    |   movel([0.069164, -1.303567, -2.624691, -0.784131, 1.570796, 1.639960],accel_mss,speed_ms,0,blend_radius_m)
    |   movel([0.068809, -1.303606, -2.624668, -0.784115, 1.570796, 1.639606],accel_mss,speed_ms,0,blend_radius_m)
    |   movel([0.068472, -1.303670, -2.624630, -0.784090, 1.570796, 1.639268],accel_mss,speed_ms,0,blend_radius_m)
    |   movel([0.068228, -1.303624, -2.624657, -0.784108, 1.570796, 1.639025],accel_mss,speed_ms,0,blend_radius_m)
    |   movel([0.068160, -1.303397, -2.624793, -0.784199, 1.570796, 1.638957],accel_mss,speed_ms,0,blend_radius_m)
    |   movel([0.067957, -1.303250, -2.624881, -0.784258, 1.570796, 1.638753],accel_mss,speed_ms,0,blend_radius_m)
    |   movel([0.067920, -1.302997, -2.625033, -0.784360, 1.570796, 1.638717],accel_mss,speed_ms,0,blend_radius_m)
    |   movel([0.068076, -1.302591, -2.625275, -0.784523, 1.570796, 1.638872],accel_mss,speed_ms,0,blend_radius_m)
    |   movel([0.068245, -1.302321, -2.625436, -0.784631, 1.570796, 1.639041],accel_mss,speed_ms,0,blend_radius_m)
    |   movel([0.068538, -1.301870, -2.625706, -0.784813, 1.570796, 1.639334],accel_mss,speed_ms,0,blend_radius_m)
    |   movel([0.068564, -1.301570, -2.625885, -0.784934, 1.570796, 1.639361],accel_mss,speed_ms,0,blend_radius_m)
    |   movel([0.068351, -1.301410, -2.625980, -0.784999, 1.570796, 1.639147],accel_mss,speed_ms,0,blend_radius_m)
    |   movel([0.068159, -1.301249, -2.626076, -0.785063, 1.570796, 1.638955],accel_mss,speed_ms,0,blend_radius_m)
    |   movel([0.068070, -1.301051, -2.626194, -0.785144, 1.570796, 1.638866],accel_mss,speed_ms,0,blend_radius_m)
    |   movel([0.067838, -1.300944, -2.626258, -0.785187, 1.570796, 1.638635],accel_mss,speed_ms,0,blend_radius_m)
    |   movel([0.067733, -1.300746, -2.626376, -0.785267, 1.570796, 1.638529],accel_mss,speed_ms,0,blend_radius_m)
    |   movel([0.067965, -1.300491, -2.626528, -0.785370, 1.570796, 1.638762],accel_mss,speed_ms,0,blend_radius_m)
    |   movel([0.068177, -1.300786, -2.626352, -0.785251, 1.570796, 1.638973],accel_mss,speed_ms,0,blend_radius_m)
    |   movel([0.068448, -1.300963, -2.626247, -0.785179, 1.570796, 1.639244],accel_mss,speed_ms,0,blend_radius_m)
    |   movel([0.068582, -1.300695, -2.626406, -0.785288, 1.570796, 1.639379],accel_mss,speed_ms,0,blend_radius_m)
    |   movel([0.068570, -1.300446, -2.626554, -0.785388, 1.570796, 1.639366],accel_mss,speed_ms,0,blend_radius_m)
    |   movel([0.068283, -1.300598, -2.626464, -0.785327, 1.570796, 1.639079],accel_mss,speed_ms,0,blend_radius_m)
    |   movel([0.068322, -1.300335, -2.626620, -0.785433, 1.570796, 1.639119],accel_mss,speed_ms,0,blend_radius_m)
    |   movel([0.068410, -1.300077, -2.626774, -0.785538, 1.570796, 1.639206],accel_mss,speed_ms,0,blend_radius_m)
    |   movel([0.068413, -1.299834, -2.626919, -0.785637, 1.570796, 1.639209],accel_mss,speed_ms,0,blend_radius_m)
    |   movel([0.068610, -1.299527, -2.627101, -0.785761, 1.570796, 1.639406],accel_mss,speed_ms,0,blend_radius_m)
    |   movel([0.068344, -1.299545, -2.627090, -0.785754, 1.570796, 1.639140],accel_mss,speed_ms,0,blend_radius_m)
    |   movel([0.068247, -1.299852, -2.626908, -0.785629, 1.570796, 1.639043],accel_mss,speed_ms,0,blend_radius_m)
    |   movel([0.068015, -1.299788, -2.626946, -0.785655, 1.570796, 1.638811],accel_mss,speed_ms,0,blend_radius_m)
    |   movel([0.068098, -1.299347, -2.627208, -0.785834, 1.570796, 1.638894],accel_mss,speed_ms,0,blend_radius_m)
    |   movel([0.068346, -1.299039, -2.627391, -0.785960, 1.570796, 1.639142],accel_mss,speed_ms,0,blend_radius_m)
    |   movel([0.068703, -1.298720, -2.627579, -0.786089, 1.570796, 1.639499],accel_mss,speed_ms,0,blend_radius_m)
    |   movel([0.069005, -1.298409, -2.627764, -0.786216, 1.570796, 1.639802],accel_mss,speed_ms,0,blend_radius_m)
    |   movel([0.068736, -1.297952, -2.628034, -0.786402, 1.570796, 1.639533],accel_mss,speed_ms,0,blend_radius_m)
    |   movel([0.068447, -1.297686, -2.628192, -0.786511, 1.570796, 1.639243],accel_mss,speed_ms,0,blend_radius_m)
    |   movel([0.068186, -1.297495, -2.628305, -0.786589, 1.570796, 1.638982],accel_mss,speed_ms,0,blend_radius_m)
    |   movel([0.068055, -1.297206, -2.628475, -0.786707, 1.570796, 1.638851],accel_mss,speed_ms,0,blend_radius_m)
    |   movel([0.068400, -1.296905, -2.628653, -0.786831, 1.570796, 1.639196],accel_mss,speed_ms,0,blend_radius_m)
    |   movel([0.068673, -1.296731, -2.628756, -0.786902, 1.570796, 1.639470],accel_mss,speed_ms,0,blend_radius_m)
    |   movel([0.068591, -1.296502, -2.628891, -0.786996, 1.570796, 1.639387],accel_mss,speed_ms,0,blend_radius_m)
    |   movel([0.068494, -1.296286, -2.629019, -0.787084, 1.570796, 1.639291],accel_mss,speed_ms,0,blend_radius_m)
    |   movel([0.068508, -1.296042, -2.629162, -0.787184, 1.570796, 1.639305],accel_mss,speed_ms,0,blend_radius_m)
    |   movel([0.068313, -1.295946, -2.629219, -0.787224, 1.570796, 1.639109],accel_mss,speed_ms,0,blend_radius_m)
    |   movel([0.068432, -1.295566, -2.629443, -0.787380, 1.570796, 1.639228],accel_mss,speed_ms,0,blend_radius_m)
    |   movel([0.068734, -1.295104, -2.629715, -0.787570, 1.570796, 1.639530],accel_mss,speed_ms,0,blend_radius_m)
    |   movel([0.069080, -1.294873, -2.629850, -0.787665, 1.570796, 1.639876],accel_mss,speed_ms,0,blend_radius_m)
    |   movel([0.069351, -1.294697, -2.629954, -0.787738, 1.570796, 1.640148],accel_mss,speed_ms,0,blend_radius_m)
    |   movel([0.069675, -1.294448, -2.630100, -0.787841, 1.570796, 1.640471],accel_mss,speed_ms,0,blend_radius_m)
    |   movel([0.069973, -1.294347, -2.630159, -0.787882, 1.570796, 1.640769],accel_mss,speed_ms,0,blend_radius_m)
    |   movel([0.070329, -1.294063, -2.630326, -0.788000, 1.570796, 1.641125],accel_mss,speed_ms,0,blend_radius_m)
    |   movel([0.070734, -1.293918, -2.630411, -0.788060, 1.570796, 1.641530],accel_mss,speed_ms,0,blend_radius_m)
    |   movel([0.070848, -1.294112, -2.630297, -0.787979, 1.570796, 1.641644],accel_mss,speed_ms,0,blend_radius_m)
    |   movel([0.070586, -1.294072, -2.630321, -0.787996, 1.570796, 1.641382],accel_mss,speed_ms,0,blend_radius_m)
    |   movel([0.070545, -1.294342, -2.630162, -0.787884, 1.570796, 1.641341],accel_mss,speed_ms,0,blend_radius_m)
    |   movel([0.070287, -1.294320, -2.630176, -0.787894, 1.570796, 1.641083],accel_mss,speed_ms,0,blend_radius_m)
    |   movel([0.070092, -1.294585, -2.630020, -0.787784, 1.570796, 1.640888],accel_mss,speed_ms,0,blend_radius_m)
    |   movel([0.069788, -1.294730, -2.629935, -0.787724, 1.570796, 1.640584],accel_mss,speed_ms,0,blend_radius_m)
    |   movel([0.070023, -1.294763, -2.629915, -0.787711, 1.570796, 1.640820],accel_mss,speed_ms,0,blend_radius_m)
    |   movel([0.070448, -1.294538, -2.630047, -0.787804, 1.570796, 1.641244],accel_mss,speed_ms,0,blend_radius_m)
    |   movel([0.070733, -1.294397, -2.630130, -0.787862, 1.570796, 1.641529],accel_mss,speed_ms,0,blend_radius_m)
    |   movel([0.071014, -1.294267, -2.630206, -0.787915, 1.570796, 1.641811],accel_mss,speed_ms,0,blend_radius_m)
    |   movel([0.071419, -1.294059, -2.630329, -0.788002, 1.570796, 1.642215],accel_mss,speed_ms,0,blend_radius_m)
    |   movel([0.071699, -1.293711, -2.630533, -0.788145, 1.570796, 1.642496],accel_mss,speed_ms,0,blend_radius_m)
    |   movel([0.071397, -1.293860, -2.630445, -0.788084, 1.570796, 1.642193],accel_mss,speed_ms,0,blend_radius_m)
    |   movel([0.071394, -1.293531, -2.630638, -0.788220, 1.570796, 1.642190],accel_mss,speed_ms,0,blend_radius_m)
    |   movel([0.071674, -1.293324, -2.630760, -0.788306, 1.570796, 1.642471],accel_mss,speed_ms,0,blend_radius_m)
    |   movel([0.072099, -1.293139, -2.630868, -0.788382, 1.570796, 1.642895],accel_mss,speed_ms,0,blend_radius_m)
    |   movel([0.072618, -1.292956, -2.630975, -0.788458, 1.570796, 1.643415],accel_mss,speed_ms,0,blend_radius_m)
    |   movel([0.072298, -1.293292, -2.630778, -0.788319, 1.570796, 1.643094],accel_mss,speed_ms,0,blend_radius_m)
    |   movel([0.072072, -1.293569, -2.630616, -0.788204, 1.570796, 1.642868],accel_mss,speed_ms,0,blend_radius_m)
    |   movel([0.072318, -1.293598, -2.630599, -0.788192, 1.570796, 1.643115],accel_mss,speed_ms,0,blend_radius_m)
    |   movel([0.072810, -1.293423, -2.630701, -0.788264, 1.570796, 1.643606],accel_mss,speed_ms,0,blend_radius_m)
    |   movel([0.073098, -1.293441, -2.630691, -0.788257, 1.570796, 1.643895],accel_mss,speed_ms,0,blend_radius_m)
    |   movel([0.073371, -1.293396, -2.630718, -0.788276, 1.570796, 1.644167],accel_mss,speed_ms,0,blend_radius_m)
    |   movel([0.073643, -1.293184, -2.630842, -0.788364, 1.570796, 1.644439],accel_mss,speed_ms,0,blend_radius_m)
    |   movel([0.073422, -1.293074, -2.630906, -0.788409, 1.570796, 1.644218],accel_mss,speed_ms,0,blend_radius_m)
    |   movel([0.073605, -1.292634, -2.631163, -0.788592, 1.570796, 1.644402],accel_mss,speed_ms,0,blend_radius_m)
    |   movel([0.074088, -1.292377, -2.631314, -0.788698, 1.570796, 1.644884],accel_mss,speed_ms,0,blend_radius_m)
    |   movel([0.074586, -1.292293, -2.631363, -0.788733, 1.570796, 1.645382],accel_mss,speed_ms,0,blend_radius_m)
    |   movel([0.075419, -1.292221, -2.631405, -0.788763, 1.570796, 1.646216],accel_mss,speed_ms,0,blend_radius_m)
    |   movel([0.075774, -1.292192, -2.631422, -0.788775, 1.570796, 1.646570],accel_mss,speed_ms,0,blend_radius_m)
    |   movel([0.076162, -1.292154, -2.631444, -0.788791, 1.570796, 1.646959],accel_mss,speed_ms,0,blend_radius_m)
    |   movel([0.076529, -1.292117, -2.631466, -0.788806, 1.570796, 1.647325],accel_mss,speed_ms,0,blend_radius_m)
    |   movel([0.076800, -1.292084, -2.631485, -0.788820, 1.570796, 1.647596],accel_mss,speed_ms,0,blend_radius_m)
    |   movel([0.077294, -1.292079, -2.631488, -0.788822, 1.570796, 1.648090],accel_mss,speed_ms,0,blend_radius_m)
    |   movel([0.077690, -1.292165, -2.631437, -0.788786, 1.570796, 1.648486],accel_mss,speed_ms,0,blend_radius_m)
    |   movel([0.078122, -1.292360, -2.631324, -0.788705, 1.570796, 1.648918],accel_mss,speed_ms,0,blend_radius_m)
    |   movel([0.078432, -1.292469, -2.631260, -0.788660, 1.570796, 1.649228],accel_mss,speed_ms,0,blend_radius_m)
    |   movel([0.078708, -1.292526, -2.631227, -0.788636, 1.570796, 1.649504],accel_mss,speed_ms,0,blend_radius_m)
    |   movel([0.079022, -1.292550, -2.631212, -0.788626, 1.570796, 1.649819],accel_mss,speed_ms,0,blend_radius_m)
    |   movel([0.079477, -1.292643, -2.631158, -0.788588, 1.570796, 1.650273],accel_mss,speed_ms,0,blend_radius_m)
    |   movel([0.080017, -1.292922, -2.630995, -0.788472, 1.570796, 1.650813],accel_mss,speed_ms,0,blend_radius_m)
    |   movel([0.080490, -1.293278, -2.630787, -0.788325, 1.570796, 1.651286],accel_mss,speed_ms,0,blend_radius_m)
    |   movel([0.080723, -1.293620, -2.630586, -0.788183, 1.570796, 1.651519],accel_mss,speed_ms,0,blend_radius_m)
    |   movel([0.080790, -1.293977, -2.630377, -0.788035, 1.570796, 1.651586],accel_mss,speed_ms,0,blend_radius_m)
    |   movel([0.080755, -1.294421, -2.630116, -0.787852, 1.570796, 1.651551],accel_mss,speed_ms,0,blend_radius_m)
    |   movel([0.080623, -1.294881, -2.629846, -0.787662, 1.570796, 1.651420],accel_mss,speed_ms,0,blend_radius_m)
    |   movel([0.080414, -1.295282, -2.629610, -0.787497, 1.570796, 1.651210],accel_mss,speed_ms,0,blend_radius_m)
    |   movel([0.080193, -1.295571, -2.629440, -0.787378, 1.570796, 1.650990],accel_mss,speed_ms,0,blend_radius_m)
    |   movel([0.079916, -1.295860, -2.629270, -0.787259, 1.570796, 1.650712],accel_mss,speed_ms,0,blend_radius_m)
    |   movel([0.079600, -1.296134, -2.629108, -0.787147, 1.570796, 1.650396],accel_mss,speed_ms,0,blend_radius_m)
    |   movel([0.079260, -1.296379, -2.628964, -0.787046, 1.570796, 1.650056],accel_mss,speed_ms,0,blend_radius_m)
    |   movel([0.079132, -1.296209, -2.629064, -0.787116, 1.570796, 1.649929],accel_mss,speed_ms,0,blend_radius_m)
    |   movel([0.078790, -1.296573, -2.628849, -0.786967, 1.570796, 1.649586],accel_mss,speed_ms,0,blend_radius_m)
    |   movel([0.078548, -1.296803, -2.628714, -0.786872, 1.570796, 1.649345],accel_mss,speed_ms,0,blend_radius_m)
    |   movel([0.078210, -1.297243, -2.628454, -0.786692, 1.570796, 1.649006],accel_mss,speed_ms,0,blend_radius_m)
    |   movel([0.078166, -1.297522, -2.628289, -0.786578, 1.570796, 1.648962],accel_mss,speed_ms,0,blend_radius_m)
    |   movel([0.078357, -1.297855, -2.628092, -0.786442, 1.570796, 1.649153],accel_mss,speed_ms,0,blend_radius_m)
    |   movel([0.078391, -1.298108, -2.627942, -0.786339, 1.570796, 1.649187],accel_mss,speed_ms,0,blend_radius_m)
    |   movel([0.078328, -1.298389, -2.627776, -0.786224, 1.570796, 1.649124],accel_mss,speed_ms,0,blend_radius_m)
    |   movel([0.078048, -1.298815, -2.627523, -0.786051, 1.570796, 1.648844],accel_mss,speed_ms,0,blend_radius_m)
    |   movel([0.078070, -1.299052, -2.627382, -0.785954, 1.570796, 1.648866],accel_mss,speed_ms,0,blend_radius_m)
    |   movel([0.077797, -1.299433, -2.627156, -0.785799, 1.570796, 1.648593],accel_mss,speed_ms,0,blend_radius_m)
    |   movel([0.077543, -1.299716, -2.626989, -0.785685, 1.570796, 1.648340],accel_mss,speed_ms,0,blend_radius_m)
    |   movel([0.077141, -1.299955, -2.626847, -0.785588, 1.570796, 1.647937],accel_mss,speed_ms,0,blend_radius_m)
    |   movel([0.076881, -1.300164, -2.626722, -0.785503, 1.570796, 1.647677],accel_mss,speed_ms,0,blend_radius_m)
    |   movel([0.076380, -1.300334, -2.626621, -0.785434, 1.570796, 1.647176],accel_mss,speed_ms,0,blend_radius_m)
    |   movel([0.076038, -1.301452, -2.625956, -0.784982, 1.570796, 1.646834],accel_mss,speed_ms,0,blend_radius_m)
    |   movel([0.075953, -1.301880, -2.625700, -0.784809, 1.570796, 1.646749],accel_mss,speed_ms,0,blend_radius_m)
    |   movel([0.075814, -1.302178, -2.625522, -0.784689, 1.570796, 1.646610],accel_mss,speed_ms,0,blend_radius_m)
    |   movel([0.075570, -1.302494, -2.625333, -0.784562, 1.570796, 1.646366],accel_mss,speed_ms,0,blend_radius_m)
    |   movel([0.075189, -1.302835, -2.625129, -0.784425, 1.570796, 1.645986],accel_mss,speed_ms,0,blend_radius_m)
    |   movel([0.074854, -1.302969, -2.625049, -0.784371, 1.570796, 1.645650],accel_mss,speed_ms,0,blend_radius_m)
    |   movel([0.074612, -1.303200, -2.624911, -0.784278, 1.570796, 1.645408],accel_mss,speed_ms,0,blend_radius_m)
    |   movel([0.074370, -1.303112, -2.624964, -0.784313, 1.570796, 1.645166],accel_mss,speed_ms,0,blend_radius_m)
    |   movel([0.074338, -1.303394, -2.624794, -0.784200, 1.570796, 1.645134],accel_mss,speed_ms,0,blend_radius_m)
    |   movel([0.073982, -1.303545, -2.624704, -0.784140, 1.570796, 1.644779],accel_mss,speed_ms,0,blend_radius_m)
    |   speed_ms = 0.003
    |   movel([0.073982, -1.289735, -2.618173, -0.804481, 1.570796, 1.644779],accel_mss,speed_ms,0,blend_radius_m)
    |   speed_ms = 1.000
    |   movel([0.073982, -1.263429, -2.604724, -0.844235, 1.570796, 1.644779],accel_mss,speed_ms,0,blend_radius_m)
    |   movel([0.076909, -1.251042, -2.611644, -0.849703, 1.570796, 1.647706],accel_mss,speed_ms,0,blend_radius_m)
    |   movel([0.076909, -1.277513, -2.625256, -0.809620, 1.570796, 1.647706],accel_mss,speed_ms,0,blend_radius_m)
    |   speed_ms = 0.003
    |   movel([0.076909, -1.287904, -2.630229, -0.794256, 1.570796, 1.647706],accel_mss,speed_ms,0,blend_radius_m)
    |   speed_ms = 0.007
    |   movel([0.076129, -1.288050, -2.630144, -0.794195, 1.570796, 1.646925],accel_mss,speed_ms,0,blend_radius_m)
    |   movel([0.075299, -1.288083, -2.630125, -0.794181, 1.570796, 1.646095],accel_mss,speed_ms,0,blend_radius_m)
    |   movel([0.074609, -1.288022, -2.630160, -0.794207, 1.570796, 1.645406],accel_mss,speed_ms,0,blend_radius_m)
    |   movel([0.074509, -1.287833, -2.630270, -0.794286, 1.570796, 1.645305],accel_mss,speed_ms,0,blend_radius_m)
    |   movel([0.074808, -1.287539, -2.630440, -0.794409, 1.570796, 1.645604],accel_mss,speed_ms,0,blend_radius_m)
    |   movel([0.075762, -1.287303, -2.630578, -0.794509, 1.570796, 1.646558],accel_mss,speed_ms,0,blend_radius_m)
    |   movel([0.076791, -1.287181, -2.630648, -0.794560, 1.570796, 1.647587],accel_mss,speed_ms,0,blend_radius_m)
    |   movel([0.077546, -1.287262, -2.630601, -0.794526, 1.570796, 1.648343],accel_mss,speed_ms,0,blend_radius_m)
    |   movel([0.077806, -1.287388, -2.630528, -0.794473, 1.570796, 1.648603],accel_mss,speed_ms,0,blend_radius_m)
    |   movel([0.077509, -1.287716, -2.630338, -0.794335, 1.570796, 1.648305],accel_mss,speed_ms,0,blend_radius_m)
    |   movel([0.076909, -1.287904, -2.630229, -0.794256, 1.570796, 1.647706],accel_mss,speed_ms,0,blend_radius_m)
    |   speed_ms = 0.003
    |   movel([0.076909, -1.291425, -2.631870, -0.789094, 1.570796, 1.647706],accel_mss,speed_ms,0,blend_radius_m)
    |   speed_ms = 0.007
    |   movel([0.076129, -1.291571, -2.631785, -0.789034, 1.570796, 1.646925],accel_mss,speed_ms,0,blend_radius_m)
    |   movel([0.075299, -1.291604, -2.631765, -0.789020, 1.570796, 1.646095],accel_mss,speed_ms,0,blend_radius_m)
    |   movel([0.074609, -1.291543, -2.631801, -0.789045, 1.570796, 1.645406],accel_mss,speed_ms,0,blend_radius_m)
    |   movel([0.074509, -1.291354, -2.631911, -0.789124, 1.570796, 1.645305],accel_mss,speed_ms,0,blend_radius_m)
    |   movel([0.074808, -1.291061, -2.632082, -0.789246, 1.570796, 1.645604],accel_mss,speed_ms,0,blend_radius_m)
    |   movel([0.075762, -1.290825, -2.632220, -0.789345, 1.570796, 1.646558],accel_mss,speed_ms,0,blend_radius_m)
    |   movel([0.076791, -1.290704, -2.632290, -0.789395, 1.570796, 1.647587],accel_mss,speed_ms,0,blend_radius_m)
    |   movel([0.077546, -1.290784, -2.632243, -0.789362, 1.570796, 1.648343],accel_mss,speed_ms,0,blend_radius_m)
    |   movel([0.077806, -1.290910, -2.632170, -0.789309, 1.570796, 1.648603],accel_mss,speed_ms,0,blend_radius_m)
    |   movel([0.077509, -1.291238, -2.631979, -0.789172, 1.570796, 1.648305],accel_mss,speed_ms,0,blend_radius_m)
    |   movel([0.076909, -1.291425, -2.631870, -0.789094, 1.570796, 1.647706],accel_mss,speed_ms,0,blend_radius_m)
    |   speed_ms = 0.003
    |   movel([0.076909, -1.277513, -2.625256, -0.809620, 1.570796, 1.647706],accel_mss,speed_ms,0,blend_radius_m)
    |   speed_ms = 1.000
    |   movel([0.076909, -1.251042, -2.611644, -0.849703, 1.570796, 1.647706],accel_mss,speed_ms,0,blend_radius_m)
    |   movel([0.077291, -1.249693, -2.612387, -0.850309, 1.570796, 1.648088],accel_mss,speed_ms,0,blend_radius_m)
    |   movel([0.077291, -1.276182, -2.626016, -0.810191, 1.570796, 1.648088],accel_mss,speed_ms,0,blend_radius_m)
    |   speed_ms = 0.003
    |   movel([0.077291, -1.286581, -2.630996, -0.794812, 1.570796, 1.648088],accel_mss,speed_ms,0,blend_radius_m)
    |   speed_ms = 0.007
    |   movel([0.076492, -1.286619, -2.630974, -0.794796, 1.570796, 1.647288],accel_mss,speed_ms,0,blend_radius_m)
    |   movel([0.075702, -1.286738, -2.630905, -0.794746, 1.570796, 1.646499],accel_mss,speed_ms,0,blend_radius_m)
    |   movel([0.075018, -1.286926, -2.630796, -0.794667, 1.570796, 1.645814],accel_mss,speed_ms,0,blend_radius_m)
    |   movel([0.074481, -1.287038, -2.630731, -0.794620, 1.570796, 1.645277],accel_mss,speed_ms,0,blend_radius_m)
    |   movel([0.074238, -1.286897, -2.630813, -0.794680, 1.570796, 1.645034],accel_mss,speed_ms,0,blend_radius_m)
    |   movel([0.074188, -1.286422, -2.631088, -0.794880, 1.570796, 1.644984],accel_mss,speed_ms,0,blend_radius_m)
    |   movel([0.074355, -1.285032, -2.631890, -0.795466, 1.570796, 1.645151],accel_mss,speed_ms,0,blend_radius_m)
    |   movel([0.074579, -1.283540, -2.632750, -0.796099, 1.570796, 1.645376],accel_mss,speed_ms,0,blend_radius_m)
    |   movel([0.074809, -1.282447, -2.633377, -0.796565, 1.570796, 1.645605],accel_mss,speed_ms,0,blend_radius_m)
    |   movel([0.075052, -1.281644, -2.633838, -0.796908, 1.570796, 1.645848],accel_mss,speed_ms,0,blend_radius_m)
    |   movel([0.075328, -1.281134, -2.634129, -0.797126, 1.570796, 1.646124],accel_mss,speed_ms,0,blend_radius_m)
    |   movel([0.076329, -1.280304, -2.634603, -0.797481, 1.570796, 1.647126],accel_mss,speed_ms,0,blend_radius_m)
    |   movel([0.078074, -1.279627, -2.634990, -0.797772, 1.570796, 1.648871],accel_mss,speed_ms,0,blend_radius_m)
    |   movel([0.079946, -1.279261, -2.635198, -0.797930, 1.570796, 1.650742],accel_mss,speed_ms,0,blend_radius_m)
    |   movel([0.081399, -1.279367, -2.635138, -0.797884, 1.570796, 1.652195],accel_mss,speed_ms,0,blend_radius_m)
    |   movel([0.081937, -1.279667, -2.634967, -0.797755, 1.570796, 1.652733],accel_mss,speed_ms,0,blend_radius_m)
    |   movel([0.082153, -1.280164, -2.634683, -0.797542, 1.570796, 1.652949],accel_mss,speed_ms,0,blend_radius_m)
    |   movel([0.082056, -1.280944, -2.634238, -0.797207, 1.570796, 1.652852],accel_mss,speed_ms,0,blend_radius_m)
    |   movel([0.081621, -1.282158, -2.633543, -0.796688, 1.570796, 1.652417],accel_mss,speed_ms,0,blend_radius_m)
    |   movel([0.081209, -1.283020, -2.633048, -0.796320, 1.570796, 1.652006],accel_mss,speed_ms,0,blend_radius_m)
    |   movel([0.080540, -1.284202, -2.632369, -0.795818, 1.570796, 1.651337],accel_mss,speed_ms,0,blend_radius_m)
    |   movel([0.079825, -1.285365, -2.631699, -0.795326, 1.570796, 1.650622],accel_mss,speed_ms,0,blend_radius_m)
    |   movel([0.079256, -1.286161, -2.631238, -0.794989, 1.570796, 1.650053],accel_mss,speed_ms,0,blend_radius_m)
    |   movel([0.078803, -1.286738, -2.630905, -0.794746, 1.570796, 1.649599],accel_mss,speed_ms,0,blend_radius_m)
    |   movel([0.078012, -1.286628, -2.630968, -0.794793, 1.570796, 1.648808],accel_mss,speed_ms,0,blend_radius_m)
    |   movel([0.077291, -1.286581, -2.630996, -0.794812, 1.570796, 1.648088],accel_mss,speed_ms,0,blend_radius_m)
    |   speed_ms = 0.003
    |   movel([0.077291, -1.290105, -2.632639, -0.789645, 1.570796, 1.648088],accel_mss,speed_ms,0,blend_radius_m)
    |   speed_ms = 0.007
    |   movel([0.076492, -1.290143, -2.632617, -0.789630, 1.570796, 1.647288],accel_mss,speed_ms,0,blend_radius_m)
    |   movel([0.075702, -1.290262, -2.632548, -0.789580, 1.570796, 1.646499],accel_mss,speed_ms,0,blend_radius_m)
    |   movel([0.075018, -1.290449, -2.632439, -0.789502, 1.570796, 1.645814],accel_mss,speed_ms,0,blend_radius_m)
    |   movel([0.074481, -1.290561, -2.632373, -0.789455, 1.570796, 1.645277],accel_mss,speed_ms,0,blend_radius_m)
    |   movel([0.074238, -1.290420, -2.632456, -0.789514, 1.570796, 1.645034],accel_mss,speed_ms,0,blend_radius_m)
    |   movel([0.074188, -1.289946, -2.632731, -0.789712, 1.570796, 1.644984],accel_mss,speed_ms,0,blend_radius_m)
    |   movel([0.074355, -1.288559, -2.633536, -0.790293, 1.570796, 1.645151],accel_mss,speed_ms,0,blend_radius_m)
    |   movel([0.074579, -1.287070, -2.634398, -0.790921, 1.570796, 1.645376],accel_mss,speed_ms,0,blend_radius_m)
    |   movel([0.074809, -1.285980, -2.635028, -0.791382, 1.570796, 1.645605],accel_mss,speed_ms,0,blend_radius_m)
    |   movel([0.075052, -1.285178, -2.635489, -0.791722, 1.570796, 1.645848],accel_mss,speed_ms,0,blend_radius_m)
    |   movel([0.075328, -1.284669, -2.635782, -0.791938, 1.570796, 1.646124],accel_mss,speed_ms,0,blend_radius_m)
    |   movel([0.076329, -1.283841, -2.636257, -0.792290, 1.570796, 1.647126],accel_mss,speed_ms,0,blend_radius_m)
    |   movel([0.078074, -1.283166, -2.636645, -0.792579, 1.570796, 1.648871],accel_mss,speed_ms,0,blend_radius_m)
    |   movel([0.079946, -1.282800, -2.636854, -0.792735, 1.570796, 1.650742],accel_mss,speed_ms,0,blend_radius_m)
    |   movel([0.081399, -1.282906, -2.636793, -0.792689, 1.570796, 1.652195],accel_mss,speed_ms,0,blend_radius_m)
    |   movel([0.081937, -1.283206, -2.636622, -0.792562, 1.570796, 1.652733],accel_mss,speed_ms,0,blend_radius_m)
    |   movel([0.082153, -1.283701, -2.636338, -0.792350, 1.570796, 1.652949],accel_mss,speed_ms,0,blend_radius_m)
    |   movel([0.082056, -1.284479, -2.635891, -0.792019, 1.570796, 1.652852],accel_mss,speed_ms,0,blend_radius_m)
    |   movel([0.081621, -1.285691, -2.635194, -0.791504, 1.570796, 1.652417],accel_mss,speed_ms,0,blend_radius_m)
    |   movel([0.081209, -1.286552, -2.634698, -0.791140, 1.570796, 1.652006],accel_mss,speed_ms,0,blend_radius_m)
    |   movel([0.080540, -1.287731, -2.634016, -0.790642, 1.570796, 1.651337],accel_mss,speed_ms,0,blend_radius_m)
    |   movel([0.079825, -1.288891, -2.633344, -0.790154, 1.570796, 1.650622],accel_mss,speed_ms,0,blend_radius_m)
    |   movel([0.079256, -1.289686, -2.632882, -0.789821, 1.570796, 1.650053],accel_mss,speed_ms,0,blend_radius_m)
    |   movel([0.078803, -1.290261, -2.632548, -0.789580, 1.570796, 1.649599],accel_mss,speed_ms,0,blend_radius_m)
    |   movel([0.078012, -1.290152, -2.632611, -0.789626, 1.570796, 1.648808],accel_mss,speed_ms,0,blend_radius_m)
    |   movel([0.077291, -1.290105, -2.632639, -0.789645, 1.570796, 1.648088],accel_mss,speed_ms,0,blend_radius_m)
    |   speed_ms = 0.003
    |   movel([0.077291, -1.276182, -2.626016, -0.810191, 1.570796, 1.648088],accel_mss,speed_ms,0,blend_radius_m)
    |   speed_ms = 1.000
    |   movel([0.077291, -1.249693, -2.612387, -0.850309, 1.570796, 1.648088],accel_mss,speed_ms,0,blend_radius_m)
    |   movel([0.079543, -1.241590, -2.616802, -0.853997, 1.570796, 1.650339],accel_mss,speed_ms,0,blend_radius_m)
    |   movel([0.079543, -1.268182, -2.630539, -0.813669, 1.570796, 1.650339],accel_mss,speed_ms,0,blend_radius_m)
    |   speed_ms = 0.003
    |   movel([0.079543, -1.278628, -2.635558, -0.798202, 1.570796, 1.650339],accel_mss,speed_ms,0,blend_radius_m)
    |   speed_ms = 0.007
    |   movel([0.079179, -1.278689, -2.635524, -0.798176, 1.570796, 1.649975],accel_mss,speed_ms,0,blend_radius_m)
    |   movel([0.078923, -1.278520, -2.635620, -0.798249, 1.570796, 1.649719],accel_mss,speed_ms,0,blend_radius_m)
    |   movel([0.078964, -1.278213, -2.635794, -0.798382, 1.570796, 1.649760],accel_mss,speed_ms,0,blend_radius_m)
    |   movel([0.079062, -1.277767, -2.636048, -0.798574, 1.570796, 1.649858],accel_mss,speed_ms,0,blend_radius_m)
    |   movel([0.079237, -1.277126, -2.636411, -0.798852, 1.570796, 1.650033],accel_mss,speed_ms,0,blend_radius_m)
    |   movel([0.079964, -1.274485, -2.637904, -0.800000, 1.570796, 1.650760],accel_mss,speed_ms,0,blend_radius_m)
    |   movel([0.080502, -1.272286, -2.639140, -0.800963, 1.570796, 1.651299],accel_mss,speed_ms,0,blend_radius_m)
    |   movel([0.080891, -1.270390, -2.640202, -0.801798, 1.570796, 1.651687],accel_mss,speed_ms,0,blend_radius_m)
    |   movel([0.081149, -1.268687, -2.641151, -0.802551, 1.570796, 1.651945],accel_mss,speed_ms,0,blend_radius_m)
    |   movel([0.081193, -1.268418, -2.641300, -0.802671, 1.570796, 1.651989],accel_mss,speed_ms,0,blend_radius_m)
    |   movel([0.081325, -1.267944, -2.641564, -0.802881, 1.570796, 1.652121],accel_mss,speed_ms,0,blend_radius_m)
    |   movel([0.081671, -1.267648, -2.641728, -0.803013, 1.570796, 1.652467],accel_mss,speed_ms,0,blend_radius_m)
    |   movel([0.082725, -1.267358, -2.641889, -0.803142, 1.570796, 1.653521],accel_mss,speed_ms,0,blend_radius_m)
    |   movel([0.083753, -1.267116, -2.642023, -0.803250, 1.570796, 1.654549],accel_mss,speed_ms,0,blend_radius_m)
    |   movel([0.084117, -1.267131, -2.642015, -0.803243, 1.570796, 1.654913],accel_mss,speed_ms,0,blend_radius_m)
    |   movel([0.084231, -1.267507, -2.641806, -0.803076, 1.570796, 1.655027],accel_mss,speed_ms,0,blend_radius_m)
    |   movel([0.084115, -1.268003, -2.641531, -0.802855, 1.570796, 1.654911],accel_mss,speed_ms,0,blend_radius_m)
    |   movel([0.083731, -1.269313, -2.640802, -0.802274, 1.570796, 1.654527],accel_mss,speed_ms,0,blend_radius_m)
    |   movel([0.082917, -1.271780, -2.639424, -0.801185, 1.570796, 1.653713],accel_mss,speed_ms,0,blend_radius_m)
    |   movel([0.081808, -1.274705, -2.637780, -0.799904, 1.570796, 1.652604],accel_mss,speed_ms,0,blend_radius_m)
    |   movel([0.080667, -1.277499, -2.636200, -0.798690, 1.570796, 1.651463],accel_mss,speed_ms,0,blend_radius_m)
    |   movel([0.080149, -1.278313, -2.635737, -0.798338, 1.570796, 1.650946],accel_mss,speed_ms,0,blend_radius_m)
    |   movel([0.079543, -1.278628, -2.635558, -0.798202, 1.570796, 1.650339],accel_mss,speed_ms,0,blend_radius_m)
    |   speed_ms = 0.003
    |   movel([0.079543, -1.282169, -2.637215, -0.793005, 1.570796, 1.650339],accel_mss,speed_ms,0,blend_radius_m)
    |   speed_ms = 0.007
    |   movel([0.079179, -1.282229, -2.637180, -0.792979, 1.570796, 1.649975],accel_mss,speed_ms,0,blend_radius_m)
    |   movel([0.078923, -1.282061, -2.637277, -0.793051, 1.570796, 1.649719],accel_mss,speed_ms,0,blend_radius_m)
    |   movel([0.078964, -1.281755, -2.637452, -0.793183, 1.570796, 1.649760],accel_mss,speed_ms,0,blend_radius_m)
    |   movel([0.079062, -1.281309, -2.637706, -0.793374, 1.570796, 1.649858],accel_mss,speed_ms,0,blend_radius_m)
    |   movel([0.079237, -1.280670, -2.638071, -0.793649, 1.570796, 1.650033],accel_mss,speed_ms,0,blend_radius_m)
    |   movel([0.079964, -1.278035, -2.639568, -0.794787, 1.570796, 1.650760],accel_mss,speed_ms,0,blend_radius_m)
    |   movel([0.080502, -1.275839, -2.640808, -0.795741, 1.570796, 1.651299],accel_mss,speed_ms,0,blend_radius_m)
    |   movel([0.080891, -1.273947, -2.641872, -0.796569, 1.570796, 1.651687],accel_mss,speed_ms,0,blend_radius_m)
    |   movel([0.081149, -1.272248, -2.642824, -0.797317, 1.570796, 1.651945],accel_mss,speed_ms,0,blend_radius_m)
    |   movel([0.081193, -1.271980, -2.642974, -0.797435, 1.570796, 1.651989],accel_mss,speed_ms,0,blend_radius_m)
    |   movel([0.081325, -1.271506, -2.643239, -0.797644, 1.570796, 1.652121],accel_mss,speed_ms,0,blend_radius_m)
    |   movel([0.081671, -1.271211, -2.643403, -0.797774, 1.570796, 1.652467],accel_mss,speed_ms,0,blend_radius_m)
    |   movel([0.082725, -1.270922, -2.643565, -0.797902, 1.570796, 1.653521],accel_mss,speed_ms,0,blend_radius_m)
    |   movel([0.083753, -1.270680, -2.643700, -0.798009, 1.570796, 1.654549],accel_mss,speed_ms,0,blend_radius_m)
    |   movel([0.084117, -1.270696, -2.643691, -0.798002, 1.570796, 1.654913],accel_mss,speed_ms,0,blend_radius_m)
    |   movel([0.084231, -1.271070, -2.643482, -0.797836, 1.570796, 1.655027],accel_mss,speed_ms,0,blend_radius_m)
    |   movel([0.084115, -1.271565, -2.643206, -0.797618, 1.570796, 1.654911],accel_mss,speed_ms,0,blend_radius_m)
    |   movel([0.083731, -1.272872, -2.642475, -0.797042, 1.570796, 1.654527],accel_mss,speed_ms,0,blend_radius_m)
    |   movel([0.082917, -1.275335, -2.641092, -0.795962, 1.570796, 1.653713],accel_mss,speed_ms,0,blend_radius_m)
    |   movel([0.081808, -1.278254, -2.639443, -0.794692, 1.570796, 1.652604],accel_mss,speed_ms,0,blend_radius_m)
    |   movel([0.080667, -1.281042, -2.637859, -0.793489, 1.570796, 1.651463],accel_mss,speed_ms,0,blend_radius_m)
    |   movel([0.080149, -1.281855, -2.637395, -0.793140, 1.570796, 1.650946],accel_mss,speed_ms,0,blend_radius_m)
    |   movel([0.079543, -1.282169, -2.637215, -0.793005, 1.570796, 1.650339],accel_mss,speed_ms,0,blend_radius_m)
    |   speed_ms = 0.003
    |   movel([0.079543, -1.268182, -2.630539, -0.813669, 1.570796, 1.650339],accel_mss,speed_ms,0,blend_radius_m)
    |   speed_ms = 1.000
    |   movel([0.079543, -1.241590, -2.616802, -0.853997, 1.570796, 1.650339],accel_mss,speed_ms,0,blend_radius_m)
    |   movel([0.082583, -1.229496, -2.623251, -0.859642, 1.570796, 1.653379],accel_mss,speed_ms,0,blend_radius_m)
    |   movel([0.082583, -1.256233, -2.637147, -0.819009, 1.570796, 1.653379],accel_mss,speed_ms,0,blend_radius_m)
    |   speed_ms = 0.003
    |   movel([0.082583, -1.266747, -2.642228, -0.803414, 1.570796, 1.653379],accel_mss,speed_ms,0,blend_radius_m)
    |   speed_ms = 0.007
    |   movel([0.081950, -1.266899, -2.642143, -0.803347, 1.570796, 1.652747],accel_mss,speed_ms,0,blend_radius_m)
    |   movel([0.081416, -1.267011, -2.642081, -0.803297, 1.570796, 1.652213],accel_mss,speed_ms,0,blend_radius_m)
    |   movel([0.080713, -1.266884, -2.642152, -0.803353, 1.570796, 1.651509],accel_mss,speed_ms,0,blend_radius_m)
    |   movel([0.080445, -1.266352, -2.642446, -0.803590, 1.570796, 1.651241],accel_mss,speed_ms,0,blend_radius_m)
    |   movel([0.080325, -1.265372, -2.642988, -0.804029, 1.570796, 1.651122],accel_mss,speed_ms,0,blend_radius_m)
    |   movel([0.080346, -1.263733, -2.643892, -0.804764, 1.570796, 1.651143],accel_mss,speed_ms,0,blend_radius_m)
    |   movel([0.080457, -1.262170, -2.644750, -0.805468, 1.570796, 1.651254],accel_mss,speed_ms,0,blend_radius_m)
    |   movel([0.080748, -1.261614, -2.645055, -0.805720, 1.570796, 1.651544],accel_mss,speed_ms,0,blend_radius_m)
    |   movel([0.081360, -1.261197, -2.645283, -0.805908, 1.570796, 1.652157],accel_mss,speed_ms,0,blend_radius_m)
    |   movel([0.083606, -1.260361, -2.645741, -0.806288, 1.570796, 1.654402],accel_mss,speed_ms,0,blend_radius_m)
    |   movel([0.084619, -1.260004, -2.645935, -0.806450, 1.570796, 1.655415],accel_mss,speed_ms,0,blend_radius_m)
    |   movel([0.085490, -1.259712, -2.646095, -0.806582, 1.570796, 1.656286],accel_mss,speed_ms,0,blend_radius_m)
    |   movel([0.086238, -1.259471, -2.646226, -0.806692, 1.570796, 1.657035],accel_mss,speed_ms,0,blend_radius_m)
    |   movel([0.086357, -1.259687, -2.646108, -0.806594, 1.570796, 1.657153],accel_mss,speed_ms,0,blend_radius_m)
    |   movel([0.086285, -1.260113, -2.645876, -0.806400, 1.570796, 1.657081],accel_mss,speed_ms,0,blend_radius_m)
    |   movel([0.086211, -1.260416, -2.645711, -0.806263, 1.570796, 1.657007],accel_mss,speed_ms,0,blend_radius_m)
    |   movel([0.086111, -1.260869, -2.645463, -0.806057, 1.570796, 1.656908],accel_mss,speed_ms,0,blend_radius_m)
    |   movel([0.086001, -1.261377, -2.645185, -0.805827, 1.570796, 1.656797],accel_mss,speed_ms,0,blend_radius_m)
    |   movel([0.085898, -1.261868, -2.644916, -0.805605, 1.570796, 1.656694],accel_mss,speed_ms,0,blend_radius_m)
    |   movel([0.085795, -1.262410, -2.644619, -0.805360, 1.570796, 1.656592],accel_mss,speed_ms,0,blend_radius_m)
    |   movel([0.085689, -1.263075, -2.644254, -0.805060, 1.570796, 1.656486],accel_mss,speed_ms,0,blend_radius_m)
    |   movel([0.085596, -1.263754, -2.643880, -0.804755, 1.570796, 1.656393],accel_mss,speed_ms,0,blend_radius_m)
    |   movel([0.085529, -1.264334, -2.643561, -0.804494, 1.570796, 1.656326],accel_mss,speed_ms,0,blend_radius_m)
    |   movel([0.085380, -1.265451, -2.642945, -0.803993, 1.570796, 1.656176],accel_mss,speed_ms,0,blend_radius_m)
    |   movel([0.085137, -1.265878, -2.642709, -0.803802, 1.570796, 1.655933],accel_mss,speed_ms,0,blend_radius_m)
    |   movel([0.084672, -1.266164, -2.642551, -0.803675, 1.570796, 1.655468],accel_mss,speed_ms,0,blend_radius_m)
    |   movel([0.083253, -1.266575, -2.642323, -0.803491, 1.570796, 1.654049],accel_mss,speed_ms,0,blend_radius_m)
    |   movel([0.082583, -1.266747, -2.642228, -0.803414, 1.570796, 1.653379],accel_mss,speed_ms,0,blend_radius_m)
    |   speed_ms = 0.003
    |   movel([0.082583, -1.270312, -2.643905, -0.798172, 1.570796, 1.653379],accel_mss,speed_ms,0,blend_radius_m)
    |   speed_ms = 0.007
    |   movel([0.081950, -1.270464, -2.643820, -0.798105, 1.570796, 1.652747],accel_mss,speed_ms,0,blend_radius_m)
    |   movel([0.081416, -1.270576, -2.643758, -0.798055, 1.570796, 1.652213],accel_mss,speed_ms,0,blend_radius_m)
    |   movel([0.080713, -1.270449, -2.643829, -0.798112, 1.570796, 1.651509],accel_mss,speed_ms,0,blend_radius_m)
    |   movel([0.080445, -1.269918, -2.644124, -0.798347, 1.570796, 1.651241],accel_mss,speed_ms,0,blend_radius_m)
    |   movel([0.080325, -1.268940, -2.644668, -0.798781, 1.570796, 1.651122],accel_mss,speed_ms,0,blend_radius_m)
    |   movel([0.080346, -1.267304, -2.645574, -0.799511, 1.570796, 1.651143],accel_mss,speed_ms,0,blend_radius_m)
    |   movel([0.080457, -1.265745, -2.646435, -0.800209, 1.570796, 1.651254],accel_mss,speed_ms,0,blend_radius_m)
    |   movel([0.080748, -1.265190, -2.646741, -0.800459, 1.570796, 1.651544],accel_mss,speed_ms,0,blend_radius_m)
    |   movel([0.081360, -1.264773, -2.646970, -0.800646, 1.570796, 1.652157],accel_mss,speed_ms,0,blend_radius_m)
    |   movel([0.083606, -1.263938, -2.647429, -0.801022, 1.570796, 1.654402],accel_mss,speed_ms,0,blend_radius_m)
    |   movel([0.084619, -1.263582, -2.647624, -0.801183, 1.570796, 1.655415],accel_mss,speed_ms,0,blend_radius_m)
    |   movel([0.085490, -1.263291, -2.647784, -0.801314, 1.570796, 1.656286],accel_mss,speed_ms,0,blend_radius_m)
    |   movel([0.086238, -1.263050, -2.647916, -0.801423, 1.570796, 1.657035],accel_mss,speed_ms,0,blend_radius_m)
    |   movel([0.086357, -1.263266, -2.647797, -0.801325, 1.570796, 1.657153],accel_mss,speed_ms,0,blend_radius_m)
    |   movel([0.086285, -1.263692, -2.647564, -0.801133, 1.570796, 1.657081],accel_mss,speed_ms,0,blend_radius_m)
    |   movel([0.086211, -1.263993, -2.647398, -0.800997, 1.570796, 1.657007],accel_mss,speed_ms,0,blend_radius_m)
    |   movel([0.086111, -1.264445, -2.647150, -0.800793, 1.570796, 1.656908],accel_mss,speed_ms,0,blend_radius_m)
    |   movel([0.086001, -1.264953, -2.646871, -0.800565, 1.570796, 1.656797],accel_mss,speed_ms,0,blend_radius_m)
    |   movel([0.085898, -1.265443, -2.646601, -0.800345, 1.570796, 1.656694],accel_mss,speed_ms,0,blend_radius_m)
    |   movel([0.085795, -1.265984, -2.646303, -0.800102, 1.570796, 1.656592],accel_mss,speed_ms,0,blend_radius_m)
    |   movel([0.085689, -1.266647, -2.645937, -0.799805, 1.570796, 1.656486],accel_mss,speed_ms,0,blend_radius_m)
    |   movel([0.085596, -1.267325, -2.645563, -0.799502, 1.570796, 1.656393],accel_mss,speed_ms,0,blend_radius_m)
    |   movel([0.085529, -1.267904, -2.645242, -0.799243, 1.570796, 1.656326],accel_mss,speed_ms,0,blend_radius_m)
    |   movel([0.085380, -1.269019, -2.644624, -0.798746, 1.570796, 1.656176],accel_mss,speed_ms,0,blend_radius_m)
    |   movel([0.085137, -1.269445, -2.644387, -0.798557, 1.570796, 1.655933],accel_mss,speed_ms,0,blend_radius_m)
    |   movel([0.084672, -1.269730, -2.644229, -0.798430, 1.570796, 1.655468],accel_mss,speed_ms,0,blend_radius_m)
    |   movel([0.083253, -1.270140, -2.644000, -0.798248, 1.570796, 1.654049],accel_mss,speed_ms,0,blend_radius_m)
    |   movel([0.082583, -1.270312, -2.643905, -0.798172, 1.570796, 1.653379],accel_mss,speed_ms,0,blend_radius_m)
    |   speed_ms = 0.003
    |   movel([0.082583, -1.256233, -2.637147, -0.819009, 1.570796, 1.653379],accel_mss,speed_ms,0,blend_radius_m)
    |   speed_ms = 1.000
    |   movel([0.082583, -1.229496, -2.623251, -0.859642, 1.570796, 1.653379],accel_mss,speed_ms,0,blend_radius_m)
    |   movel([0.092310, -1.229064, -2.623478, -0.859847, 1.570796, 1.663107],accel_mss,speed_ms,0,blend_radius_m)
    |   movel([0.092310, -1.255806, -2.637380, -0.819203, 1.570796, 1.663107],accel_mss,speed_ms,0,blend_radius_m)
    |   speed_ms = 0.003
    |   movel([0.092310, -1.266323, -2.642463, -0.803604, 1.570796, 1.663107],accel_mss,speed_ms,0,blend_radius_m)
    |   speed_ms = 0.007
    |   movel([0.093445, -1.265797, -2.642754, -0.803839, 1.570796, 1.664242],accel_mss,speed_ms,0,blend_radius_m)
    |   movel([0.094363, -1.265473, -2.642933, -0.803984, 1.570796, 1.665160],accel_mss,speed_ms,0,blend_radius_m)
    |   movel([0.094630, -1.265516, -2.642909, -0.803964, 1.570796, 1.665426],accel_mss,speed_ms,0,blend_radius_m)
    |   movel([0.094539, -1.265873, -2.642711, -0.803804, 1.570796, 1.665336],accel_mss,speed_ms,0,blend_radius_m)
    |   movel([0.094064, -1.266107, -2.642582, -0.803700, 1.570796, 1.664861],accel_mss,speed_ms,0,blend_radius_m)
    |   movel([0.093493, -1.266293, -2.642479, -0.803617, 1.570796, 1.664289],accel_mss,speed_ms,0,blend_radius_m)
    |   movel([0.092792, -1.266495, -2.642367, -0.803527, 1.570796, 1.663589],accel_mss,speed_ms,0,blend_radius_m)
    |   movel([0.092422, -1.266550, -2.642337, -0.803502, 1.570796, 1.663219],accel_mss,speed_ms,0,blend_radius_m)
    |   movel([0.092310, -1.266323, -2.642463, -0.803604, 1.570796, 1.663107],accel_mss,speed_ms,0,blend_radius_m)
    |   speed_ms = 0.003
    |   movel([0.092310, -1.269888, -2.644140, -0.798360, 1.570796, 1.663107],accel_mss,speed_ms,0,blend_radius_m)
    |   speed_ms = 0.007
    |   movel([0.093445, -1.269364, -2.644432, -0.798593, 1.570796, 1.664242],accel_mss,speed_ms,0,blend_radius_m)
    |   movel([0.094363, -1.269040, -2.644612, -0.798737, 1.570796, 1.665160],accel_mss,speed_ms,0,blend_radius_m)
    |   movel([0.094630, -1.269083, -2.644588, -0.798718, 1.570796, 1.665426],accel_mss,speed_ms,0,blend_radius_m)
    |   movel([0.094539, -1.269440, -2.644390, -0.798559, 1.570796, 1.665336],accel_mss,speed_ms,0,blend_radius_m)
    |   movel([0.094064, -1.269673, -2.644260, -0.798456, 1.570796, 1.664861],accel_mss,speed_ms,0,blend_radius_m)
    |   movel([0.093493, -1.269859, -2.644157, -0.798373, 1.570796, 1.664289],accel_mss,speed_ms,0,blend_radius_m)
    |   movel([0.092792, -1.270060, -2.644045, -0.798284, 1.570796, 1.663589],accel_mss,speed_ms,0,blend_radius_m)
    |   movel([0.092422, -1.270115, -2.644014, -0.798259, 1.570796, 1.663219],accel_mss,speed_ms,0,blend_radius_m)
    |   movel([0.092310, -1.269888, -2.644140, -0.798360, 1.570796, 1.663107],accel_mss,speed_ms,0,blend_radius_m)
    |   speed_ms = 0.003
    |   movel([0.092310, -1.255806, -2.637380, -0.819203, 1.570796, 1.663107],accel_mss,speed_ms,0,blend_radius_m)
    |   speed_ms = 1.000
    |   movel([0.092310, -1.229064, -2.623478, -0.859847, 1.570796, 1.663107],accel_mss,speed_ms,0,blend_radius_m)
    |   movel([0.099561, -1.230071, -2.622948, -0.859370, 1.570796, 1.670358],accel_mss,speed_ms,0,blend_radius_m)
    |   movel([0.099561, -1.256801, -2.636837, -0.818751, 1.570796, 1.670358],accel_mss,speed_ms,0,blend_radius_m)
    |   speed_ms = 0.003
    |   movel([0.099561, -1.267312, -2.641914, -0.803162, 1.570796, 1.670358],accel_mss,speed_ms,0,blend_radius_m)
    |   speed_ms = 0.007
    |   movel([0.099947, -1.267089, -2.642038, -0.803262, 1.570796, 1.670743],accel_mss,speed_ms,0,blend_radius_m)
    |   movel([0.100597, -1.266887, -2.642150, -0.803352, 1.570796, 1.671393],accel_mss,speed_ms,0,blend_radius_m)
    |   movel([0.101348, -1.266671, -2.642270, -0.803448, 1.570796, 1.672144],accel_mss,speed_ms,0,blend_radius_m)
    |   movel([0.101677, -1.266608, -2.642305, -0.803476, 1.570796, 1.672473],accel_mss,speed_ms,0,blend_radius_m)
    |   movel([0.101808, -1.266783, -2.642208, -0.803398, 1.570796, 1.672604],accel_mss,speed_ms,0,blend_radius_m)
    |   movel([0.101464, -1.267006, -2.642084, -0.803299, 1.570796, 1.672260],accel_mss,speed_ms,0,blend_radius_m)
    |   movel([0.101097, -1.267158, -2.642000, -0.803231, 1.570796, 1.671893],accel_mss,speed_ms,0,blend_radius_m)
    |   movel([0.100604, -1.267336, -2.641901, -0.803152, 1.570796, 1.671400],accel_mss,speed_ms,0,blend_radius_m)
    |   movel([0.099927, -1.267559, -2.641777, -0.803052, 1.570796, 1.670723],accel_mss,speed_ms,0,blend_radius_m)
    |   movel([0.099533, -1.267588, -2.641761, -0.803040, 1.570796, 1.670330],accel_mss,speed_ms,0,blend_radius_m)
    |   movel([0.099561, -1.267312, -2.641914, -0.803162, 1.570796, 1.670358],accel_mss,speed_ms,0,blend_radius_m)
    |   speed_ms = 0.003
    |   movel([0.099561, -1.270876, -2.643590, -0.797922, 1.570796, 1.670358],accel_mss,speed_ms,0,blend_radius_m)
    |   speed_ms = 0.007
    |   movel([0.099947, -1.270654, -2.643714, -0.798021, 1.570796, 1.670743],accel_mss,speed_ms,0,blend_radius_m)
    |   movel([0.100597, -1.270452, -2.643827, -0.798110, 1.570796, 1.671393],accel_mss,speed_ms,0,blend_radius_m)
    |   movel([0.101348, -1.270236, -2.643947, -0.798206, 1.570796, 1.672144],accel_mss,speed_ms,0,blend_radius_m)
    |   movel([0.101677, -1.270173, -2.643982, -0.798234, 1.570796, 1.672473],accel_mss,speed_ms,0,blend_radius_m)
    |   movel([0.101808, -1.270348, -2.643885, -0.798156, 1.570796, 1.672604],accel_mss,speed_ms,0,blend_radius_m)
    |   movel([0.101464, -1.270571, -2.643761, -0.798058, 1.570796, 1.672260],accel_mss,speed_ms,0,blend_radius_m)
    |   movel([0.101097, -1.270722, -2.643676, -0.797991, 1.570796, 1.671893],accel_mss,speed_ms,0,blend_radius_m)
    |   movel([0.100604, -1.270900, -2.643577, -0.797912, 1.570796, 1.671400],accel_mss,speed_ms,0,blend_radius_m)
    |   movel([0.099927, -1.271123, -2.643453, -0.797813, 1.570796, 1.670723],accel_mss,speed_ms,0,blend_radius_m)
    |   movel([0.099533, -1.271151, -2.643437, -0.797801, 1.570796, 1.670330],accel_mss,speed_ms,0,blend_radius_m)
    |   movel([0.099561, -1.270876, -2.643590, -0.797922, 1.570796, 1.670358],accel_mss,speed_ms,0,blend_radius_m)
    |   speed_ms = 0.003
    |   movel([0.099561, -1.256801, -2.636837, -0.818751, 1.570796, 1.670358],accel_mss,speed_ms,0,blend_radius_m)
    |   speed_ms = 1.000
    |   movel([0.099561, -1.230071, -2.622948, -0.859370, 1.570796, 1.670358],accel_mss,speed_ms,0,blend_radius_m)
    |   movel([0.099464, -1.229425, -2.623288, -0.859676, 1.570796, 1.670261],accel_mss,speed_ms,0,blend_radius_m)
    |   movel([0.099464, -1.256163, -2.637185, -0.819041, 1.570796, 1.670261],accel_mss,speed_ms,0,blend_radius_m)
    |   speed_ms = 0.003
    |   movel([0.099464, -1.266678, -2.642266, -0.803445, 1.570796, 1.670261],accel_mss,speed_ms,0,blend_radius_m)
    |   speed_ms = 0.007
    |   movel([0.099864, -1.266398, -2.642421, -0.803570, 1.570796, 1.670661],accel_mss,speed_ms,0,blend_radius_m)
    |   movel([0.100140, -1.265931, -2.642679, -0.803779, 1.570796, 1.670936],accel_mss,speed_ms,0,blend_radius_m)
    |   movel([0.100356, -1.265081, -2.643149, -0.804159, 1.570796, 1.671153],accel_mss,speed_ms,0,blend_radius_m)
    |   movel([0.100640, -1.263246, -2.644160, -0.804983, 1.570796, 1.671436],accel_mss,speed_ms,0,blend_radius_m)
    |   movel([0.100880, -1.261605, -2.645060, -0.805724, 1.570796, 1.671677],accel_mss,speed_ms,0,blend_radius_m)
    |   movel([0.101009, -1.260957, -2.645415, -0.806017, 1.570796, 1.671805],accel_mss,speed_ms,0,blend_radius_m)
    |   movel([0.101145, -1.260582, -2.645620, -0.806187, 1.570796, 1.671942],accel_mss,speed_ms,0,blend_radius_m)
    |   movel([0.101358, -1.260292, -2.645778, -0.806319, 1.570796, 1.672154],accel_mss,speed_ms,0,blend_radius_m)
    |   movel([0.101658, -1.260042, -2.645915, -0.806432, 1.570796, 1.672454],accel_mss,speed_ms,0,blend_radius_m)
    |   movel([0.102128, -1.259955, -2.645962, -0.806472, 1.570796, 1.672924],accel_mss,speed_ms,0,blend_radius_m)
    |   movel([0.102340, -1.260116, -2.645874, -0.806399, 1.570796, 1.673136],accel_mss,speed_ms,0,blend_radius_m)
    |   movel([0.102446, -1.260348, -2.645747, -0.806293, 1.570796, 1.673242],accel_mss,speed_ms,0,blend_radius_m)
    |   movel([0.102458, -1.260728, -2.645540, -0.806121, 1.570796, 1.673254],accel_mss,speed_ms,0,blend_radius_m)
    |   movel([0.102379, -1.261416, -2.645164, -0.805809, 1.570796, 1.673176],accel_mss,speed_ms,0,blend_radius_m)
    |   movel([0.102123, -1.263031, -2.644278, -0.805080, 1.570796, 1.672919],accel_mss,speed_ms,0,blend_radius_m)
    |   movel([0.101853, -1.264772, -2.643319, -0.804297, 1.570796, 1.672649],accel_mss,speed_ms,0,blend_radius_m)
    |   movel([0.101798, -1.265520, -2.642906, -0.803962, 1.570796, 1.672594],accel_mss,speed_ms,0,blend_radius_m)
    |   movel([0.101884, -1.265846, -2.642726, -0.803816, 1.570796, 1.672681],accel_mss,speed_ms,0,blend_radius_m)
    |   movel([0.102127, -1.265892, -2.642701, -0.803796, 1.570796, 1.672923],accel_mss,speed_ms,0,blend_radius_m)
    |   movel([0.102418, -1.265924, -2.642683, -0.803782, 1.570796, 1.673214],accel_mss,speed_ms,0,blend_radius_m)
    |   movel([0.102637, -1.266057, -2.642610, -0.803722, 1.570796, 1.673433],accel_mss,speed_ms,0,blend_radius_m)
    |   movel([0.102685, -1.266335, -2.642456, -0.803598, 1.570796, 1.673481],accel_mss,speed_ms,0,blend_radius_m)
    |   movel([0.102479, -1.266979, -2.642099, -0.803311, 1.570796, 1.673275],accel_mss,speed_ms,0,blend_radius_m)
    |   movel([0.102314, -1.267259, -2.641944, -0.803186, 1.570796, 1.673111],accel_mss,speed_ms,0,blend_radius_m)
    |   movel([0.101871, -1.267582, -2.641764, -0.803042, 1.570796, 1.672667],accel_mss,speed_ms,0,blend_radius_m)
    |   movel([0.101580, -1.267799, -2.641644, -0.802946, 1.570796, 1.672376],accel_mss,speed_ms,0,blend_radius_m)
    |   movel([0.101261, -1.268211, -2.641416, -0.802763, 1.570796, 1.672057],accel_mss,speed_ms,0,blend_radius_m)
    |   movel([0.100848, -1.268752, -2.641115, -0.802523, 1.570796, 1.671644],accel_mss,speed_ms,0,blend_radius_m)
    |   movel([0.100469, -1.268999, -2.640977, -0.802413, 1.570796, 1.671265],accel_mss,speed_ms,0,blend_radius_m)
    |   movel([0.100136, -1.268960, -2.640999, -0.802430, 1.570796, 1.670932],accel_mss,speed_ms,0,blend_radius_m)
    |   movel([0.099864, -1.268617, -2.641190, -0.802582, 1.570796, 1.670660],accel_mss,speed_ms,0,blend_radius_m)
    |   movel([0.099641, -1.268371, -2.641327, -0.802692, 1.570796, 1.670438],accel_mss,speed_ms,0,blend_radius_m)
    |   movel([0.099334, -1.268343, -2.641342, -0.802704, 1.570796, 1.670130],accel_mss,speed_ms,0,blend_radius_m)
    |   movel([0.098951, -1.268375, -2.641324, -0.802690, 1.570796, 1.669747],accel_mss,speed_ms,0,blend_radius_m)
    |   movel([0.098703, -1.268278, -2.641378, -0.802733, 1.570796, 1.669500],accel_mss,speed_ms,0,blend_radius_m)
    |   movel([0.098605, -1.268048, -2.641506, -0.802835, 1.570796, 1.669401],accel_mss,speed_ms,0,blend_radius_m)
    |   movel([0.098652, -1.267700, -2.641699, -0.802990, 1.570796, 1.669448],accel_mss,speed_ms,0,blend_radius_m)
    |   movel([0.098799, -1.267292, -2.641925, -0.803171, 1.570796, 1.669595],accel_mss,speed_ms,0,blend_radius_m)
    |   movel([0.098967, -1.267010, -2.642082, -0.803297, 1.570796, 1.669764],accel_mss,speed_ms,0,blend_radius_m)
    |   movel([0.099464, -1.266678, -2.642266, -0.803445, 1.570796, 1.670261],accel_mss,speed_ms,0,blend_radius_m)
    |   speed_ms = 0.003
    |   movel([0.099464, -1.270243, -2.643943, -0.798203, 1.570796, 1.670261],accel_mss,speed_ms,0,blend_radius_m)
    |   speed_ms = 0.007
    |   movel([0.099864, -1.269963, -2.644099, -0.798327, 1.570796, 1.670661],accel_mss,speed_ms,0,blend_radius_m)
    |   movel([0.100140, -1.269497, -2.644358, -0.798534, 1.570796, 1.670936],accel_mss,speed_ms,0,blend_radius_m)
    |   movel([0.100356, -1.268649, -2.644829, -0.798911, 1.570796, 1.671153],accel_mss,speed_ms,0,blend_radius_m)
    |   movel([0.100640, -1.266818, -2.645843, -0.799728, 1.570796, 1.671436],accel_mss,speed_ms,0,blend_radius_m)
    |   movel([0.100880, -1.265181, -2.646746, -0.800463, 1.570796, 1.671677],accel_mss,speed_ms,0,blend_radius_m)
    |   movel([0.101009, -1.264534, -2.647102, -0.800754, 1.570796, 1.671805],accel_mss,speed_ms,0,blend_radius_m)
    |   movel([0.101145, -1.264159, -2.647307, -0.800923, 1.570796, 1.671942],accel_mss,speed_ms,0,blend_radius_m)
    |   movel([0.101358, -1.263870, -2.647466, -0.801053, 1.570796, 1.672154],accel_mss,speed_ms,0,blend_radius_m)
    |   movel([0.101658, -1.263620, -2.647603, -0.801166, 1.570796, 1.672454],accel_mss,speed_ms,0,blend_radius_m)
    |   movel([0.102128, -1.263533, -2.647651, -0.801205, 1.570796, 1.672924],accel_mss,speed_ms,0,blend_radius_m)
    |   movel([0.102340, -1.263694, -2.647563, -0.801132, 1.570796, 1.673136],accel_mss,speed_ms,0,blend_radius_m)
    |   movel([0.102446, -1.263926, -2.647435, -0.801028, 1.570796, 1.673242],accel_mss,speed_ms,0,blend_radius_m)
    |   movel([0.102458, -1.264305, -2.647228, -0.800857, 1.570796, 1.673254],accel_mss,speed_ms,0,blend_radius_m)
    |   movel([0.102379, -1.264992, -2.646850, -0.800548, 1.570796, 1.673176],accel_mss,speed_ms,0,blend_radius_m)
    |   movel([0.102123, -1.266603, -2.645961, -0.799825, 1.570796, 1.672919],accel_mss,speed_ms,0,blend_radius_m)
    |   movel([0.101853, -1.268341, -2.645000, -0.799048, 1.570796, 1.672649],accel_mss,speed_ms,0,blend_radius_m)
    |   movel([0.101798, -1.269088, -2.644586, -0.798716, 1.570796, 1.672594],accel_mss,speed_ms,0,blend_radius_m)
    |   movel([0.101884, -1.269413, -2.644405, -0.798571, 1.570796, 1.672681],accel_mss,speed_ms,0,blend_radius_m)
    |   movel([0.102127, -1.269459, -2.644379, -0.798551, 1.570796, 1.672923],accel_mss,speed_ms,0,blend_radius_m)
    |   movel([0.102418, -1.269491, -2.644362, -0.798537, 1.570796, 1.673214],accel_mss,speed_ms,0,blend_radius_m)
    |   movel([0.102637, -1.269624, -2.644288, -0.798478, 1.570796, 1.673433],accel_mss,speed_ms,0,blend_radius_m)
    |   movel([0.102685, -1.269900, -2.644134, -0.798355, 1.570796, 1.673481],accel_mss,speed_ms,0,blend_radius_m)
    |   movel([0.102479, -1.270544, -2.643776, -0.798070, 1.570796, 1.673275],accel_mss,speed_ms,0,blend_radius_m)
    |   movel([0.102314, -1.270823, -2.643620, -0.797946, 1.570796, 1.673111],accel_mss,speed_ms,0,blend_radius_m)
    |   movel([0.101871, -1.271146, -2.643440, -0.797803, 1.570796, 1.672667],accel_mss,speed_ms,0,blend_radius_m)
    |   movel([0.101580, -1.271362, -2.643319, -0.797707, 1.570796, 1.672376],accel_mss,speed_ms,0,blend_radius_m)
    |   movel([0.101261, -1.271773, -2.643090, -0.797526, 1.570796, 1.672057],accel_mss,speed_ms,0,blend_radius_m)
    |   movel([0.100848, -1.272313, -2.642788, -0.797288, 1.570796, 1.671644],accel_mss,speed_ms,0,blend_radius_m)
    |   movel([0.100469, -1.272559, -2.642650, -0.797179, 1.570796, 1.671265],accel_mss,speed_ms,0,blend_radius_m)
    |   movel([0.100136, -1.272520, -2.642672, -0.797197, 1.570796, 1.670932],accel_mss,speed_ms,0,blend_radius_m)
    |   movel([0.099864, -1.272178, -2.642863, -0.797347, 1.570796, 1.670660],accel_mss,speed_ms,0,blend_radius_m)
    |   movel([0.099641, -1.271932, -2.643001, -0.797456, 1.570796, 1.670438],accel_mss,speed_ms,0,blend_radius_m)
    |   movel([0.099334, -1.271905, -2.643016, -0.797468, 1.570796, 1.670130],accel_mss,speed_ms,0,blend_radius_m)
    |   movel([0.098951, -1.271937, -2.642998, -0.797454, 1.570796, 1.669747],accel_mss,speed_ms,0,blend_radius_m)
    |   movel([0.098703, -1.271840, -2.643053, -0.797497, 1.570796, 1.669500],accel_mss,speed_ms,0,blend_radius_m)
    |   movel([0.098605, -1.271610, -2.643181, -0.797598, 1.570796, 1.669401],accel_mss,speed_ms,0,blend_radius_m)
    |   movel([0.098652, -1.271263, -2.643375, -0.797751, 1.570796, 1.669448],accel_mss,speed_ms,0,blend_radius_m)
    |   movel([0.098799, -1.270856, -2.643602, -0.797931, 1.570796, 1.669595],accel_mss,speed_ms,0,blend_radius_m)
    |   movel([0.098967, -1.270575, -2.643758, -0.798056, 1.570796, 1.669764],accel_mss,speed_ms,0,blend_radius_m)
    |   movel([0.099464, -1.270243, -2.643943, -0.798203, 1.570796, 1.670261],accel_mss,speed_ms,0,blend_radius_m)
    |   speed_ms = 0.003
    |   movel([0.099464, -1.256163, -2.637185, -0.819041, 1.570796, 1.670261],accel_mss,speed_ms,0,blend_radius_m)
    |   speed_ms = 1.000
    |   movel([0.099464, -1.229425, -2.623288, -0.859676, 1.570796, 1.670261],accel_mss,speed_ms,0,blend_radius_m)
    |   movel([0.085805, -1.233581, -2.621092, -0.857716, 1.570796, 1.656601],accel_mss,speed_ms,0,blend_radius_m)
    |   movel([0.085805, -1.260270, -2.634934, -0.817185, 1.570796, 1.656601],accel_mss,speed_ms,0,blend_radius_m)
    |   speed_ms = 0.003
    |   movel([0.085805, -1.270762, -2.639994, -0.801634, 1.570796, 1.656601],accel_mss,speed_ms,0,blend_radius_m)
    |   speed_ms = 0.007
    |   movel([0.086070, -1.265880, -2.642708, -0.803802, 1.570796, 1.656867],accel_mss,speed_ms,0,blend_radius_m)
    |   movel([0.086295, -1.263990, -2.643750, -0.804649, 1.570796, 1.657092],accel_mss,speed_ms,0,blend_radius_m)
    |   movel([0.086599, -1.262035, -2.644825, -0.805530, 1.570796, 1.657396],accel_mss,speed_ms,0,blend_radius_m)
    |   movel([0.086929, -1.260286, -2.645781, -0.806321, 1.570796, 1.657725],accel_mss,speed_ms,0,blend_radius_m)
    |   movel([0.087180, -1.259543, -2.646187, -0.806659, 1.570796, 1.657976],accel_mss,speed_ms,0,blend_radius_m)
    |   movel([0.087885, -1.258813, -2.646585, -0.806992, 1.570796, 1.658681],accel_mss,speed_ms,0,blend_radius_m)
    |   movel([0.089726, -1.257950, -2.647054, -0.807385, 1.570796, 1.660522],accel_mss,speed_ms,0,blend_radius_m)
    |   movel([0.092956, -1.256741, -2.647709, -0.807938, 1.570796, 1.663752],accel_mss,speed_ms,0,blend_radius_m)
    |   movel([0.099627, -1.254504, -2.648919, -0.808966, 1.570796, 1.670423],accel_mss,speed_ms,0,blend_radius_m)
    |   movel([0.109598, -1.251283, -2.650649, -0.810457, 1.570796, 1.680394],accel_mss,speed_ms,0,blend_radius_m)
    |   movel([0.114228, -1.249893, -2.651392, -0.811104, 1.570796, 1.685025],accel_mss,speed_ms,0,blend_radius_m)
    |   movel([0.116925, -1.249198, -2.651762, -0.811429, 1.570796, 1.687721],accel_mss,speed_ms,0,blend_radius_m)
    |   movel([0.117802, -1.249298, -2.651709, -0.811382, 1.570796, 1.688598],accel_mss,speed_ms,0,blend_radius_m)
    |   movel([0.118115, -1.249499, -2.651602, -0.811289, 1.570796, 1.688912],accel_mss,speed_ms,0,blend_radius_m)
    |   movel([0.117518, -1.253510, -2.649454, -0.809425, 1.570796, 1.688314],accel_mss,speed_ms,0,blend_radius_m)
    |   movel([0.117200, -1.255550, -2.648354, -0.808485, 1.570796, 1.687996],accel_mss,speed_ms,0,blend_radius_m)
    |   movel([0.116930, -1.257094, -2.647518, -0.807777, 1.570796, 1.687727],accel_mss,speed_ms,0,blend_radius_m)
    |   movel([0.116660, -1.258388, -2.646816, -0.807185, 1.570796, 1.687457],accel_mss,speed_ms,0,blend_radius_m)
    |   movel([0.116358, -1.259620, -2.646145, -0.806624, 1.570796, 1.687154],accel_mss,speed_ms,0,blend_radius_m)
    |   movel([0.115266, -1.263334, -2.644111, -0.804944, 1.570796, 1.686062],accel_mss,speed_ms,0,blend_radius_m)
    |   movel([0.114094, -1.266630, -2.642293, -0.803466, 1.570796, 1.684890],accel_mss,speed_ms,0,blend_radius_m)
    |   movel([0.112789, -1.269640, -2.640620, -0.802129, 1.570796, 1.683586],accel_mss,speed_ms,0,blend_radius_m)
    |   movel([0.111308, -1.272482, -2.639030, -0.800877, 1.570796, 1.682104],accel_mss,speed_ms,0,blend_radius_m)
    |   movel([0.109151, -1.275877, -2.637118, -0.799394, 1.570796, 1.679948],accel_mss,speed_ms,0,blend_radius_m)
    |   movel([0.106892, -1.278659, -2.635541, -0.798189, 1.570796, 1.677688],accel_mss,speed_ms,0,blend_radius_m)
    |   movel([0.104397, -1.280981, -2.634217, -0.797191, 1.570796, 1.675193],accel_mss,speed_ms,0,blend_radius_m)
    |   movel([0.101531, -1.282996, -2.633062, -0.796331, 1.570796, 1.672327],accel_mss,speed_ms,0,blend_radius_m)
    |   movel([0.100843, -1.283390, -2.632836, -0.796163, 1.570796, 1.671639],accel_mss,speed_ms,0,blend_radius_m)
    |   movel([0.100214, -1.283699, -2.632658, -0.796032, 1.570796, 1.671010],accel_mss,speed_ms,0,blend_radius_m)
    |   movel([0.099441, -1.284018, -2.632475, -0.795896, 1.570796, 1.670237],accel_mss,speed_ms,0,blend_radius_m)
    |   movel([0.098221, -1.284469, -2.632215, -0.795705, 1.570796, 1.669018],accel_mss,speed_ms,0,blend_radius_m)
    |   movel([0.096957, -1.284915, -2.631958, -0.795516, 1.570796, 1.667754],accel_mss,speed_ms,0,blend_radius_m)
    |   movel([0.096211, -1.285147, -2.631824, -0.795418, 1.570796, 1.667007],accel_mss,speed_ms,0,blend_radius_m)
    |   movel([0.095602, -1.285283, -2.631746, -0.795360, 1.570796, 1.666399],accel_mss,speed_ms,0,blend_radius_m)
    |   movel([0.094884, -1.285382, -2.631688, -0.795318, 1.570796, 1.665680],accel_mss,speed_ms,0,blend_radius_m)
    |   movel([0.092619, -1.285335, -2.631716, -0.795338, 1.570796, 1.663416],accel_mss,speed_ms,0,blend_radius_m)
    |   movel([0.090657, -1.284691, -2.632087, -0.795611, 1.570796, 1.661453],accel_mss,speed_ms,0,blend_radius_m)
    |   movel([0.089028, -1.283443, -2.632805, -0.796140, 1.570796, 1.659824],accel_mss,speed_ms,0,blend_radius_m)
    |   movel([0.087745, -1.281605, -2.633860, -0.796924, 1.570796, 1.658541],accel_mss,speed_ms,0,blend_radius_m)
    |   movel([0.086658, -1.278724, -2.635504, -0.798161, 1.570796, 1.657455],accel_mss,speed_ms,0,blend_radius_m)
    |   movel([0.086008, -1.275074, -2.637572, -0.799743, 1.570796, 1.656804],accel_mss,speed_ms,0,blend_radius_m)
    |   movel([0.085805, -1.270762, -2.639994, -0.801634, 1.570796, 1.656601],accel_mss,speed_ms,0,blend_radius_m)
    |   speed_ms = 0.003
    |   movel([0.085805, -1.274319, -2.641664, -0.796406, 1.570796, 1.656601],accel_mss,speed_ms,0,blend_radius_m)
    |   speed_ms = 0.007
    |   movel([0.086070, -1.269446, -2.644386, -0.798556, 1.570796, 1.656867],accel_mss,speed_ms,0,blend_radius_m)
    |   movel([0.086295, -1.267560, -2.645432, -0.799396, 1.570796, 1.657092],accel_mss,speed_ms,0,blend_radius_m)
    |   movel([0.086599, -1.265609, -2.646510, -0.800270, 1.570796, 1.657396],accel_mss,speed_ms,0,blend_radius_m)
    |   movel([0.086929, -1.263864, -2.647469, -0.801056, 1.570796, 1.657725],accel_mss,speed_ms,0,blend_radius_m)
    |   movel([0.087180, -1.263122, -2.647876, -0.801391, 1.570796, 1.657976],accel_mss,speed_ms,0,blend_radius_m)
    |   movel([0.087885, -1.262393, -2.648275, -0.801720, 1.570796, 1.658681],accel_mss,speed_ms,0,blend_radius_m)
    |   movel([0.089726, -1.261532, -2.648746, -0.802111, 1.570796, 1.660522],accel_mss,speed_ms,0,blend_radius_m)
    |   movel([0.092956, -1.260326, -2.649404, -0.802659, 1.570796, 1.663752],accel_mss,speed_ms,0,blend_radius_m)
    |   movel([0.099627, -1.258093, -2.650617, -0.803680, 1.570796, 1.670423],accel_mss,speed_ms,0,blend_radius_m)
    |   movel([0.109598, -1.254878, -2.652352, -0.805159, 1.570796, 1.680394],accel_mss,speed_ms,0,blend_radius_m)
    |   movel([0.114228, -1.253491, -2.653097, -0.805801, 1.570796, 1.685025],accel_mss,speed_ms,0,blend_radius_m)
    |   movel([0.116925, -1.252797, -2.653469, -0.806123, 1.570796, 1.687721],accel_mss,speed_ms,0,blend_radius_m)
    |   movel([0.117802, -1.252896, -2.653416, -0.806077, 1.570796, 1.688598],accel_mss,speed_ms,0,blend_radius_m)
    |   movel([0.118115, -1.253097, -2.653308, -0.805984, 1.570796, 1.688912],accel_mss,speed_ms,0,blend_radius_m)
    |   movel([0.117518, -1.257101, -2.651153, -0.804135, 1.570796, 1.688314],accel_mss,speed_ms,0,blend_radius_m)
    |   movel([0.117200, -1.259137, -2.650050, -0.803202, 1.570796, 1.687996],accel_mss,speed_ms,0,blend_radius_m)
    |   movel([0.116930, -1.260678, -2.649212, -0.802499, 1.570796, 1.687727],accel_mss,speed_ms,0,blend_radius_m)
    |   movel([0.116660, -1.261969, -2.648507, -0.801913, 1.570796, 1.687457],accel_mss,speed_ms,0,blend_radius_m)
    |   movel([0.116358, -1.263199, -2.647834, -0.801356, 1.570796, 1.687154],accel_mss,speed_ms,0,blend_radius_m)
    |   movel([0.115266, -1.266906, -2.645794, -0.799689, 1.570796, 1.686062],accel_mss,speed_ms,0,blend_radius_m)
    |   movel([0.114094, -1.270195, -2.643970, -0.798224, 1.570796, 1.684890],accel_mss,speed_ms,0,blend_radius_m)
    |   movel([0.112789, -1.273199, -2.642292, -0.796898, 1.570796, 1.683586],accel_mss,speed_ms,0,blend_radius_m)
    |   movel([0.111308, -1.276036, -2.640697, -0.795656, 1.570796, 1.682104],accel_mss,speed_ms,0,blend_radius_m)
    |   movel([0.109151, -1.279423, -2.638780, -0.794186, 1.570796, 1.679948],accel_mss,speed_ms,0,blend_radius_m)
    |   movel([0.106892, -1.282199, -2.637198, -0.792992, 1.570796, 1.677688],accel_mss,speed_ms,0,blend_radius_m)
    |   movel([0.104397, -1.284517, -2.635870, -0.792003, 1.570796, 1.675193],accel_mss,speed_ms,0,blend_radius_m)
    |   movel([0.101531, -1.286527, -2.634712, -0.791150, 1.570796, 1.672327],accel_mss,speed_ms,0,blend_radius_m)
    |   movel([0.100843, -1.286920, -2.634485, -0.790984, 1.570796, 1.671639],accel_mss,speed_ms,0,blend_radius_m)
    |   movel([0.100214, -1.287229, -2.634306, -0.790853, 1.570796, 1.671010],accel_mss,speed_ms,0,blend_radius_m)
    |   movel([0.099441, -1.287548, -2.634122, -0.790719, 1.570796, 1.670237],accel_mss,speed_ms,0,blend_radius_m)
    |   movel([0.098221, -1.287998, -2.633862, -0.790530, 1.570796, 1.669018],accel_mss,speed_ms,0,blend_radius_m)
    |   movel([0.096957, -1.288442, -2.633604, -0.790343, 1.570796, 1.667754],accel_mss,speed_ms,0,blend_radius_m)
    |   movel([0.096211, -1.288674, -2.633470, -0.790245, 1.570796, 1.667007],accel_mss,speed_ms,0,blend_radius_m)
    |   movel([0.095602, -1.288810, -2.633391, -0.790188, 1.570796, 1.666399],accel_mss,speed_ms,0,blend_radius_m)
    |   movel([0.094884, -1.288909, -2.633334, -0.790147, 1.570796, 1.665680],accel_mss,speed_ms,0,blend_radius_m)
    |   movel([0.092619, -1.288862, -2.633361, -0.790166, 1.570796, 1.663416],accel_mss,speed_ms,0,blend_radius_m)
    |   movel([0.090657, -1.288219, -2.633734, -0.790437, 1.570796, 1.661453],accel_mss,speed_ms,0,blend_radius_m)
    |   movel([0.089028, -1.286974, -2.634454, -0.790961, 1.570796, 1.659824],accel_mss,speed_ms,0,blend_radius_m)
    |   movel([0.087745, -1.285140, -2.635511, -0.791738, 1.570796, 1.658541],accel_mss,speed_ms,0,blend_radius_m)
    |   movel([0.086658, -1.282264, -2.637161, -0.792964, 1.570796, 1.657455],accel_mss,speed_ms,0,blend_radius_m)
    |   movel([0.086008, -1.278622, -2.639235, -0.794532, 1.570796, 1.656804],accel_mss,speed_ms,0,blend_radius_m)
    |   movel([0.085805, -1.274319, -2.641664, -0.796406, 1.570796, 1.656601],accel_mss,speed_ms,0,blend_radius_m)
    |   speed_ms = 0.003
    |   movel([0.085805, -1.260270, -2.634934, -0.817185, 1.570796, 1.656601],accel_mss,speed_ms,0,blend_radius_m)
    |   speed_ms = 1.000
    |   movel([0.085805, -1.233581, -2.621092, -0.857716, 1.570796, 1.656601],accel_mss,speed_ms,0,blend_radius_m)
    |   movel([0.090276, -1.249111, -2.612707, -0.850572, 1.570796, 1.661072],accel_mss,speed_ms,0,blend_radius_m)
    |   movel([0.090276, -1.275607, -2.626344, -0.810438, 1.570796, 1.661072],accel_mss,speed_ms,0,blend_radius_m)
    |   speed_ms = 0.003
    |   movel([0.090276, -1.286010, -2.631326, -0.795053, 1.570796, 1.661072],accel_mss,speed_ms,0,blend_radius_m)
    |   speed_ms = 0.007
    |   speed_ms = 0.003
    |   movel([0.090276, -1.289535, -2.632970, -0.789884, 1.570796, 1.661072],accel_mss,speed_ms,0,blend_radius_m)
    |   speed_ms = 0.007
    |   speed_ms = 0.003
    |   movel([0.090276, -1.275607, -2.626344, -0.810438, 1.570796, 1.661072],accel_mss,speed_ms,0,blend_radius_m)
    |   speed_ms = 1.000
    |   movel([0.090276, -1.249111, -2.612707, -0.850572, 1.570796, 1.661072],accel_mss,speed_ms,0,blend_radius_m)
    |   movel([0.090517, -1.275491, -2.626410, -0.810488, 1.570796, 1.661314],accel_mss,speed_ms,0,blend_radius_m)
    |   speed_ms = 0.003
    |   movel([0.090517, -1.285894, -2.631393, -0.795102, 1.570796, 1.661314],accel_mss,speed_ms,0,blend_radius_m)
    |   speed_ms = 0.007
    |   movel([0.090760, -1.285956, -2.631357, -0.795076, 1.570796, 1.661556],accel_mss,speed_ms,0,blend_radius_m)
    |   movel([0.091359, -1.285967, -2.631351, -0.795071, 1.570796, 1.662155],accel_mss,speed_ms,0,blend_radius_m)
    |   movel([0.091835, -1.286012, -2.631325, -0.795052, 1.570796, 1.662631],accel_mss,speed_ms,0,blend_radius_m)
    |   movel([0.092380, -1.286070, -2.631291, -0.795028, 1.570796, 1.663177],accel_mss,speed_ms,0,blend_radius_m)
    |   movel([0.092996, -1.286119, -2.631263, -0.795007, 1.570796, 1.663793],accel_mss,speed_ms,0,blend_radius_m)
    |   movel([0.093656, -1.286137, -2.631252, -0.795000, 1.570796, 1.664452],accel_mss,speed_ms,0,blend_radius_m)
    |   movel([0.094270, -1.286128, -2.631258, -0.795004, 1.570796, 1.665066],accel_mss,speed_ms,0,blend_radius_m)
    |   movel([0.094742, -1.286082, -2.631284, -0.795023, 1.570796, 1.665538],accel_mss,speed_ms,0,blend_radius_m)
    |   movel([0.097078, -1.285558, -2.631587, -0.795244, 1.570796, 1.667875],accel_mss,speed_ms,0,blend_radius_m)
    |   movel([0.099439, -1.284682, -2.632092, -0.795615, 1.570796, 1.670236],accel_mss,speed_ms,0,blend_radius_m)
    |   movel([0.101784, -1.283471, -2.632789, -0.796129, 1.570796, 1.672581],accel_mss,speed_ms,0,blend_radius_m)
    |   movel([0.104076, -1.281941, -2.633667, -0.796780, 1.570796, 1.674873],accel_mss,speed_ms,0,blend_radius_m)
    |   movel([0.104777, -1.281474, -2.633935, -0.796980, 1.570796, 1.675573],accel_mss,speed_ms,0,blend_radius_m)
    |   movel([0.105551, -1.281055, -2.634174, -0.797159, 1.570796, 1.676347],accel_mss,speed_ms,0,blend_radius_m)
    |   movel([0.106203, -1.280776, -2.634334, -0.797279, 1.570796, 1.676999],accel_mss,speed_ms,0,blend_radius_m)
    |   movel([0.106394, -1.280924, -2.634249, -0.797216, 1.570796, 1.677190],accel_mss,speed_ms,0,blend_radius_m)
    |   movel([0.106666, -1.280931, -2.634245, -0.797212, 1.570796, 1.677462],accel_mss,speed_ms,0,blend_radius_m)
    |   movel([0.106922, -1.280639, -2.634412, -0.797338, 1.570796, 1.677719],accel_mss,speed_ms,0,blend_radius_m)
    |   movel([0.107235, -1.280554, -2.634461, -0.797374, 1.570796, 1.678032],accel_mss,speed_ms,0,blend_radius_m)
    |   movel([0.106944, -1.280659, -2.634401, -0.797329, 1.570796, 1.677741],accel_mss,speed_ms,0,blend_radius_m)
    |   movel([0.107092, -1.280910, -2.634257, -0.797222, 1.570796, 1.677889],accel_mss,speed_ms,0,blend_radius_m)
    |   movel([0.107397, -1.280825, -2.634306, -0.797258, 1.570796, 1.678194],accel_mss,speed_ms,0,blend_radius_m)
    |   movel([0.107675, -1.280853, -2.634290, -0.797246, 1.570796, 1.678471],accel_mss,speed_ms,0,blend_radius_m)
    |   movel([0.107807, -1.281013, -2.634199, -0.797178, 1.570796, 1.678603],accel_mss,speed_ms,0,blend_radius_m)
    |   movel([0.108113, -1.280823, -2.634307, -0.797259, 1.570796, 1.678910],accel_mss,speed_ms,0,blend_radius_m)
    |   movel([0.107859, -1.280759, -2.634344, -0.797287, 1.570796, 1.678655],accel_mss,speed_ms,0,blend_radius_m)
    |   movel([0.107530, -1.280639, -2.634412, -0.797338, 1.570796, 1.678327],accel_mss,speed_ms,0,blend_radius_m)
    |   movel([0.108087, -1.280418, -2.634538, -0.797433, 1.570796, 1.678883],accel_mss,speed_ms,0,blend_radius_m)
    |   movel([0.108555, -1.280456, -2.634517, -0.797416, 1.570796, 1.679351],accel_mss,speed_ms,0,blend_radius_m)
    |   movel([0.109052, -1.280655, -2.634403, -0.797331, 1.570796, 1.679849],accel_mss,speed_ms,0,blend_radius_m)
    |   movel([0.109447, -1.280935, -2.634243, -0.797211, 1.570796, 1.680244],accel_mss,speed_ms,0,blend_radius_m)
    |   movel([0.109568, -1.281224, -2.634078, -0.797087, 1.570796, 1.680365],accel_mss,speed_ms,0,blend_radius_m)
    |   movel([0.109559, -1.281633, -2.633843, -0.796912, 1.570796, 1.680355],accel_mss,speed_ms,0,blend_radius_m)
    |   movel([0.109485, -1.281925, -2.633676, -0.796787, 1.570796, 1.680281],accel_mss,speed_ms,0,blend_radius_m)
    |   movel([0.109326, -1.282211, -2.633512, -0.796665, 1.570796, 1.680122],accel_mss,speed_ms,0,blend_radius_m)
    |   movel([0.109017, -1.282599, -2.633290, -0.796500, 1.570796, 1.679813],accel_mss,speed_ms,0,blend_radius_m)
    |   movel([0.108778, -1.282857, -2.633142, -0.796390, 1.570796, 1.679574],accel_mss,speed_ms,0,blend_radius_m)
    |   movel([0.108466, -1.283158, -2.632969, -0.796262, 1.570796, 1.679263],accel_mss,speed_ms,0,blend_radius_m)
    |   movel([0.108137, -1.283451, -2.632801, -0.796137, 1.570796, 1.678934],accel_mss,speed_ms,0,blend_radius_m)
    |   movel([0.107842, -1.283689, -2.632664, -0.796036, 1.570796, 1.678638],accel_mss,speed_ms,0,blend_radius_m)
    |   movel([0.107121, -1.284217, -2.632360, -0.795812, 1.570796, 1.677917],accel_mss,speed_ms,0,blend_radius_m)
    |   movel([0.106892, -1.284128, -2.632412, -0.795850, 1.570796, 1.677688],accel_mss,speed_ms,0,blend_radius_m)
    |   movel([0.107390, -1.283544, -2.632747, -0.796097, 1.570796, 1.678187],accel_mss,speed_ms,0,blend_radius_m)
    |   movel([0.107724, -1.283168, -2.632963, -0.796257, 1.570796, 1.678521],accel_mss,speed_ms,0,blend_radius_m)
    |   movel([0.107352, -1.283374, -2.632845, -0.796170, 1.570796, 1.678148],accel_mss,speed_ms,0,blend_radius_m)
    |   movel([0.107190, -1.283667, -2.632676, -0.796045, 1.570796, 1.677986],accel_mss,speed_ms,0,blend_radius_m)
    |   movel([0.106820, -1.283786, -2.632609, -0.795995, 1.570796, 1.677616],accel_mss,speed_ms,0,blend_radius_m)
    |   movel([0.106429, -1.284151, -2.632398, -0.795840, 1.570796, 1.677225],accel_mss,speed_ms,0,blend_radius_m)
    |   movel([0.106409, -1.284430, -2.632238, -0.795722, 1.570796, 1.677205],accel_mss,speed_ms,0,blend_radius_m)
    |   movel([0.106162, -1.284337, -2.632291, -0.795761, 1.570796, 1.676958],accel_mss,speed_ms,0,blend_radius_m)
    |   movel([0.105915, -1.284689, -2.632088, -0.795612, 1.570796, 1.676711],accel_mss,speed_ms,0,blend_radius_m)
    |   movel([0.106042, -1.284980, -2.631921, -0.795489, 1.570796, 1.676838],accel_mss,speed_ms,0,blend_radius_m)
    |   movel([0.106016, -1.285267, -2.631755, -0.795367, 1.570796, 1.676812],accel_mss,speed_ms,0,blend_radius_m)
    |   movel([0.106280, -1.285257, -2.631760, -0.795371, 1.570796, 1.677077],accel_mss,speed_ms,0,blend_radius_m)
    |   movel([0.106205, -1.285570, -2.631580, -0.795239, 1.570796, 1.677002],accel_mss,speed_ms,0,blend_radius_m)
    |   movel([0.106244, -1.285829, -2.631431, -0.795130, 1.570796, 1.677041],accel_mss,speed_ms,0,blend_radius_m)
    |   movel([0.106515, -1.285998, -2.631333, -0.795058, 1.570796, 1.677311],accel_mss,speed_ms,0,blend_radius_m)
    |   movel([0.106800, -1.285814, -2.631439, -0.795136, 1.570796, 1.677596],accel_mss,speed_ms,0,blend_radius_m)
    |   movel([0.106483, -1.285854, -2.631416, -0.795119, 1.570796, 1.677280],accel_mss,speed_ms,0,blend_radius_m)
    |   movel([0.106363, -1.285576, -2.631576, -0.795236, 1.570796, 1.677160],accel_mss,speed_ms,0,blend_radius_m)
    |   movel([0.106782, -1.285404, -2.631676, -0.795309, 1.570796, 1.677578],accel_mss,speed_ms,0,blend_radius_m)
    |   movel([0.106980, -1.285541, -2.631597, -0.795251, 1.570796, 1.677777],accel_mss,speed_ms,0,blend_radius_m)
    |   movel([0.107145, -1.285783, -2.631457, -0.795149, 1.570796, 1.677941],accel_mss,speed_ms,0,blend_radius_m)
    |   movel([0.107185, -1.286078, -2.631287, -0.795025, 1.570796, 1.677981],accel_mss,speed_ms,0,blend_radius_m)
    |   movel([0.107094, -1.286383, -2.631110, -0.794896, 1.570796, 1.677891],accel_mss,speed_ms,0,blend_radius_m)
    |   movel([0.106889, -1.286660, -2.630950, -0.794779, 1.570796, 1.677685],accel_mss,speed_ms,0,blend_radius_m)
    |   movel([0.106730, -1.287021, -2.630741, -0.794627, 1.570796, 1.677527],accel_mss,speed_ms,0,blend_radius_m)
    |   movel([0.106361, -1.287438, -2.630499, -0.794452, 1.570796, 1.677157],accel_mss,speed_ms,0,blend_radius_m)
    |   movel([0.106023, -1.287751, -2.630318, -0.794321, 1.570796, 1.676819],accel_mss,speed_ms,0,blend_radius_m)
    |   movel([0.105735, -1.287964, -2.630194, -0.794231, 1.570796, 1.676531],accel_mss,speed_ms,0,blend_radius_m)
    |   movel([0.105337, -1.288150, -2.630086, -0.794153, 1.570796, 1.676133],accel_mss,speed_ms,0,blend_radius_m)
    |   movel([0.104955, -1.288387, -2.629948, -0.794054, 1.570796, 1.675752],accel_mss,speed_ms,0,blend_radius_m)
    |   movel([0.104548, -1.288586, -2.629833, -0.793970, 1.570796, 1.675345],accel_mss,speed_ms,0,blend_radius_m)
    |   movel([0.103748, -1.288777, -2.629722, -0.793890, 1.570796, 1.674544],accel_mss,speed_ms,0,blend_radius_m)
    |   movel([0.103011, -1.289005, -2.629589, -0.793795, 1.570796, 1.673807],accel_mss,speed_ms,0,blend_radius_m)
    |   movel([0.102355, -1.289248, -2.629448, -0.793694, 1.570796, 1.673152],accel_mss,speed_ms,0,blend_radius_m)
    |   movel([0.101965, -1.289540, -2.629278, -0.793572, 1.570796, 1.672761],accel_mss,speed_ms,0,blend_radius_m)
    |   movel([0.101499, -1.289699, -2.629185, -0.793505, 1.570796, 1.672295],accel_mss,speed_ms,0,blend_radius_m)
    |   movel([0.101150, -1.289866, -2.629088, -0.793435, 1.570796, 1.671947],accel_mss,speed_ms,0,blend_radius_m)
    |   movel([0.100675, -1.289847, -2.629098, -0.793443, 1.570796, 1.671471],accel_mss,speed_ms,0,blend_radius_m)
    |   movel([0.100391, -1.289890, -2.629073, -0.793425, 1.570796, 1.671188],accel_mss,speed_ms,0,blend_radius_m)
    |   movel([0.100053, -1.290183, -2.628903, -0.793303, 1.570796, 1.670849],accel_mss,speed_ms,0,blend_radius_m)
    |   movel([0.100321, -1.290199, -2.628893, -0.793297, 1.570796, 1.671118],accel_mss,speed_ms,0,blend_radius_m)
    |   movel([0.100651, -1.290151, -2.628921, -0.793317, 1.570796, 1.671448],accel_mss,speed_ms,0,blend_radius_m)
    |   movel([0.101031, -1.290134, -2.628931, -0.793324, 1.570796, 1.671827],accel_mss,speed_ms,0,blend_radius_m)
    |   movel([0.101319, -1.290099, -2.628952, -0.793338, 1.570796, 1.672116],accel_mss,speed_ms,0,blend_radius_m)
    |   movel([0.101619, -1.290054, -2.628978, -0.793357, 1.570796, 1.672416],accel_mss,speed_ms,0,blend_radius_m)
    |   movel([0.102043, -1.289977, -2.629023, -0.793389, 1.570796, 1.672840],accel_mss,speed_ms,0,blend_radius_m)
    |   movel([0.101987, -1.289743, -2.629159, -0.793487, 1.570796, 1.672784],accel_mss,speed_ms,0,blend_radius_m)
    |   movel([0.102373, -1.289772, -2.629142, -0.793475, 1.570796, 1.673169],accel_mss,speed_ms,0,blend_radius_m)
    |   movel([0.102475, -1.289975, -2.629024, -0.793390, 1.570796, 1.673271],accel_mss,speed_ms,0,blend_radius_m)
    |   movel([0.102816, -1.289921, -2.629056, -0.793413, 1.570796, 1.673613],accel_mss,speed_ms,0,blend_radius_m)
    |   movel([0.103104, -1.289884, -2.629077, -0.793428, 1.570796, 1.673901],accel_mss,speed_ms,0,blend_radius_m)
    |   movel([0.103382, -1.289827, -2.629110, -0.793452, 1.570796, 1.674178],accel_mss,speed_ms,0,blend_radius_m)
    |   movel([0.103678, -1.289588, -2.629250, -0.793552, 1.570796, 1.674474],accel_mss,speed_ms,0,blend_radius_m)
    |   movel([0.103359, -1.289746, -2.629157, -0.793485, 1.570796, 1.674155],accel_mss,speed_ms,0,blend_radius_m)
    |   movel([0.103194, -1.289619, -2.629232, -0.793539, 1.570796, 1.673991],accel_mss,speed_ms,0,blend_radius_m)
    |   movel([0.103230, -1.289311, -2.629411, -0.793667, 1.570796, 1.674026],accel_mss,speed_ms,0,blend_radius_m)
    |   movel([0.103561, -1.289000, -2.629592, -0.793797, 1.570796, 1.674358],accel_mss,speed_ms,0,blend_radius_m)
    |   movel([0.103869, -1.288936, -2.629629, -0.793824, 1.570796, 1.674665],accel_mss,speed_ms,0,blend_radius_m)
    |   movel([0.103902, -1.289178, -2.629488, -0.793723, 1.570796, 1.674699],accel_mss,speed_ms,0,blend_radius_m)
    |   movel([0.104086, -1.289372, -2.629376, -0.793642, 1.570796, 1.674882],accel_mss,speed_ms,0,blend_radius_m)
    |   movel([0.104470, -1.289572, -2.629259, -0.793558, 1.570796, 1.675266],accel_mss,speed_ms,0,blend_radius_m)
    |   movel([0.104480, -1.289893, -2.629072, -0.793424, 1.570796, 1.675276],accel_mss,speed_ms,0,blend_radius_m)
    |   movel([0.104166, -1.289990, -2.629015, -0.793384, 1.570796, 1.674962],accel_mss,speed_ms,0,blend_radius_m)
    |   movel([0.103943, -1.289929, -2.629051, -0.793409, 1.570796, 1.674739],accel_mss,speed_ms,0,blend_radius_m)
    |   movel([0.103724, -1.289790, -2.629132, -0.793467, 1.570796, 1.674520],accel_mss,speed_ms,0,blend_radius_m)
    |   movel([0.103804, -1.290067, -2.628970, -0.793352, 1.570796, 1.674600],accel_mss,speed_ms,0,blend_radius_m)
    |   movel([0.103792, -1.290462, -2.628740, -0.793187, 1.570796, 1.674589],accel_mss,speed_ms,0,blend_radius_m)
    |   movel([0.103523, -1.290823, -2.628529, -0.793037, 1.570796, 1.674319],accel_mss,speed_ms,0,blend_radius_m)
    |   movel([0.103297, -1.291104, -2.628365, -0.792920, 1.570796, 1.674094],accel_mss,speed_ms,0,blend_radius_m)
    |   movel([0.102982, -1.291173, -2.628325, -0.792892, 1.570796, 1.673778],accel_mss,speed_ms,0,blend_radius_m)
    |   movel([0.102668, -1.291475, -2.628148, -0.792766, 1.570796, 1.673465],accel_mss,speed_ms,0,blend_radius_m)
    |   movel([0.102281, -1.291681, -2.628027, -0.792680, 1.570796, 1.673077],accel_mss,speed_ms,0,blend_radius_m)
    |   movel([0.101902, -1.291838, -2.627935, -0.792615, 1.570796, 1.672698],accel_mss,speed_ms,0,blend_radius_m)
    |   movel([0.101557, -1.291976, -2.627854, -0.792558, 1.570796, 1.672353],accel_mss,speed_ms,0,blend_radius_m)
    |   movel([0.101243, -1.292105, -2.627779, -0.792505, 1.570796, 1.672039],accel_mss,speed_ms,0,blend_radius_m)
    |   movel([0.101286, -1.292331, -2.627647, -0.792411, 1.570796, 1.672083],accel_mss,speed_ms,0,blend_radius_m)
    |   movel([0.100997, -1.292480, -2.627559, -0.792350, 1.570796, 1.671793],accel_mss,speed_ms,0,blend_radius_m)
    |   movel([0.100718, -1.292440, -2.627583, -0.792366, 1.570796, 1.671514],accel_mss,speed_ms,0,blend_radius_m)
    |   movel([0.100425, -1.292566, -2.627509, -0.792314, 1.570796, 1.671222],accel_mss,speed_ms,0,blend_radius_m)
    |   movel([0.099331, -1.293071, -2.627213, -0.792105, 1.570796, 1.670127],accel_mss,speed_ms,0,blend_radius_m)
    |   movel([0.097242, -1.293784, -2.626794, -0.791811, 1.570796, 1.668038],accel_mss,speed_ms,0,blend_radius_m)
    |   movel([0.095038, -1.294457, -2.626398, -0.791534, 1.570796, 1.665834],accel_mss,speed_ms,0,blend_radius_m)
    |   movel([0.093267, -1.294893, -2.626141, -0.791355, 1.570796, 1.664064],accel_mss,speed_ms,0,blend_radius_m)
    |   movel([0.092796, -1.295002, -2.626077, -0.791310, 1.570796, 1.663592],accel_mss,speed_ms,0,blend_radius_m)
    |   movel([0.092505, -1.295072, -2.626035, -0.791282, 1.570796, 1.663301],accel_mss,speed_ms,0,blend_radius_m)
    |   movel([0.092006, -1.295190, -2.625966, -0.791233, 1.570796, 1.662802],accel_mss,speed_ms,0,blend_radius_m)
    |   movel([0.091686, -1.295204, -2.625958, -0.791227, 1.570796, 1.662483],accel_mss,speed_ms,0,blend_radius_m)
    |   movel([0.091516, -1.295043, -2.626052, -0.791293, 1.570796, 1.662312],accel_mss,speed_ms,0,blend_radius_m)
    |   movel([0.090908, -1.295099, -2.626020, -0.791271, 1.570796, 1.661704],accel_mss,speed_ms,0,blend_radius_m)
    |   movel([0.091012, -1.295287, -2.625909, -0.791193, 1.570796, 1.661808],accel_mss,speed_ms,0,blend_radius_m)
    |   movel([0.091131, -1.295453, -2.625811, -0.791125, 1.570796, 1.661927],accel_mss,speed_ms,0,blend_radius_m)
    |   movel([0.091380, -1.295526, -2.625768, -0.791095, 1.570796, 1.662176],accel_mss,speed_ms,0,blend_radius_m)
    |   movel([0.091703, -1.295529, -2.625766, -0.791094, 1.570796, 1.662500],accel_mss,speed_ms,0,blend_radius_m)
    |   movel([0.091970, -1.295280, -2.625913, -0.791196, 1.570796, 1.662766],accel_mss,speed_ms,0,blend_radius_m)
    |   movel([0.092331, -1.295302, -2.625900, -0.791187, 1.570796, 1.663127],accel_mss,speed_ms,0,blend_radius_m)
    |   movel([0.092659, -1.295213, -2.625953, -0.791224, 1.570796, 1.663455],accel_mss,speed_ms,0,blend_radius_m)
    |   movel([0.092762, -1.295396, -2.625845, -0.791149, 1.570796, 1.663559],accel_mss,speed_ms,0,blend_radius_m)
    |   movel([0.092991, -1.295457, -2.625808, -0.791124, 1.570796, 1.663787],accel_mss,speed_ms,0,blend_radius_m)
    |   movel([0.093296, -1.295278, -2.625914, -0.791197, 1.570796, 1.664092],accel_mss,speed_ms,0,blend_radius_m)
    |   movel([0.093554, -1.295264, -2.625922, -0.791203, 1.570796, 1.664350],accel_mss,speed_ms,0,blend_radius_m)
    |   movel([0.093259, -1.295524, -2.625769, -0.791096, 1.570796, 1.664056],accel_mss,speed_ms,0,blend_radius_m)
    |   movel([0.092956, -1.295608, -2.625719, -0.791062, 1.570796, 1.663753],accel_mss,speed_ms,0,blend_radius_m)
    |   movel([0.092691, -1.295566, -2.625744, -0.791079, 1.570796, 1.663487],accel_mss,speed_ms,0,blend_radius_m)
    |   movel([0.092356, -1.295474, -2.625799, -0.791117, 1.570796, 1.663152],accel_mss,speed_ms,0,blend_radius_m)
    |   movel([0.092063, -1.295519, -2.625772, -0.791098, 1.570796, 1.662859],accel_mss,speed_ms,0,blend_radius_m)
    |   movel([0.091652, -1.295639, -2.625701, -0.791049, 1.570796, 1.662448],accel_mss,speed_ms,0,blend_radius_m)
    |   movel([0.091327, -1.295728, -2.625649, -0.791013, 1.570796, 1.662123],accel_mss,speed_ms,0,blend_radius_m)
    |   movel([0.091035, -1.295784, -2.625615, -0.790989, 1.570796, 1.661832],accel_mss,speed_ms,0,blend_radius_m)
    |   movel([0.090721, -1.295828, -2.625590, -0.790972, 1.570796, 1.661517],accel_mss,speed_ms,0,blend_radius_m)
    |   movel([0.090684, -1.295590, -2.625730, -0.791069, 1.570796, 1.661480],accel_mss,speed_ms,0,blend_radius_m)
    |   movel([0.090510, -1.295461, -2.625806, -0.791122, 1.570796, 1.661306],accel_mss,speed_ms,0,blend_radius_m)
    |   movel([0.090188, -1.295575, -2.625739, -0.791075, 1.570796, 1.660984],accel_mss,speed_ms,0,blend_radius_m)
    |   movel([0.090012, -1.295435, -2.625821, -0.791133, 1.570796, 1.660808],accel_mss,speed_ms,0,blend_radius_m)
    |   movel([0.089943, -1.295224, -2.625946, -0.791219, 1.570796, 1.660739],accel_mss,speed_ms,0,blend_radius_m)
    |   movel([0.089712, -1.295174, -2.625976, -0.791240, 1.570796, 1.660509],accel_mss,speed_ms,0,blend_radius_m)
    |   movel([0.089970, -1.294932, -2.626118, -0.791339, 1.570796, 1.660766],accel_mss,speed_ms,0,blend_radius_m)
    |   movel([0.090285, -1.294888, -2.626144, -0.791357, 1.570796, 1.661081],accel_mss,speed_ms,0,blend_radius_m)
    |   movel([0.090132, -1.295178, -2.625973, -0.791238, 1.570796, 1.660928],accel_mss,speed_ms,0,blend_radius_m)
    |   movel([0.090205, -1.295458, -2.625808, -0.791123, 1.570796, 1.661001],accel_mss,speed_ms,0,blend_radius_m)
    |   movel([0.090261, -1.295173, -2.625976, -0.791240, 1.570796, 1.661057],accel_mss,speed_ms,0,blend_radius_m)
    |   movel([0.090563, -1.295048, -2.626049, -0.791291, 1.570796, 1.661359],accel_mss,speed_ms,0,blend_radius_m)
    |   movel([0.090470, -1.294836, -2.626175, -0.791378, 1.570796, 1.661266],accel_mss,speed_ms,0,blend_radius_m)
    |   movel([0.090383, -1.294562, -2.626336, -0.791491, 1.570796, 1.661179],accel_mss,speed_ms,0,blend_radius_m)
    |   movel([0.090678, -1.294319, -2.626479, -0.791591, 1.570796, 1.661474],accel_mss,speed_ms,0,blend_radius_m)
    |   movel([0.090825, -1.293986, -2.626675, -0.791728, 1.570796, 1.661621],accel_mss,speed_ms,0,blend_radius_m)
    |   movel([0.090518, -1.294183, -2.626559, -0.791647, 1.570796, 1.661314],accel_mss,speed_ms,0,blend_radius_m)
    |   movel([0.090290, -1.294420, -2.626420, -0.791549, 1.570796, 1.661086],accel_mss,speed_ms,0,blend_radius_m)
    |   movel([0.090113, -1.294706, -2.626251, -0.791432, 1.570796, 1.660910],accel_mss,speed_ms,0,blend_radius_m)
    |   movel([0.089804, -1.294774, -2.626211, -0.791404, 1.570796, 1.660600],accel_mss,speed_ms,0,blend_radius_m)
    |   movel([0.089954, -1.294457, -2.626398, -0.791534, 1.570796, 1.660750],accel_mss,speed_ms,0,blend_radius_m)
    |   movel([0.090167, -1.294184, -2.626558, -0.791646, 1.570796, 1.660963],accel_mss,speed_ms,0,blend_radius_m)
    |   movel([0.090457, -1.293839, -2.626762, -0.791789, 1.570796, 1.661253],accel_mss,speed_ms,0,blend_radius_m)
    |   movel([0.090350, -1.293548, -2.626933, -0.791909, 1.570796, 1.661146],accel_mss,speed_ms,0,blend_radius_m)
    |   movel([0.090002, -1.293462, -2.626983, -0.791944, 1.570796, 1.660798],accel_mss,speed_ms,0,blend_radius_m)
    |   movel([0.089628, -1.293427, -2.627004, -0.791959, 1.570796, 1.660424],accel_mss,speed_ms,0,blend_radius_m)
    |   movel([0.089304, -1.293469, -2.626979, -0.791941, 1.570796, 1.660101],accel_mss,speed_ms,0,blend_radius_m)
    |   movel([0.089032, -1.293425, -2.627005, -0.791959, 1.570796, 1.659829],accel_mss,speed_ms,0,blend_radius_m)
    |   movel([0.088749, -1.293465, -2.626981, -0.791943, 1.570796, 1.659546],accel_mss,speed_ms,0,blend_radius_m)
    |   movel([0.088519, -1.293407, -2.627015, -0.791966, 1.570796, 1.659315],accel_mss,speed_ms,0,blend_radius_m)
    |   movel([0.088260, -1.293283, -2.627088, -0.792018, 1.570796, 1.659057],accel_mss,speed_ms,0,blend_radius_m)
    |   movel([0.087984, -1.293094, -2.627199, -0.792096, 1.570796, 1.658780],accel_mss,speed_ms,0,blend_radius_m)
    |   movel([0.087838, -1.292892, -2.627318, -0.792179, 1.570796, 1.658634],accel_mss,speed_ms,0,blend_radius_m)
    |   movel([0.087930, -1.292619, -2.627478, -0.792292, 1.570796, 1.658726],accel_mss,speed_ms,0,blend_radius_m)
    |   movel([0.088018, -1.292324, -2.627651, -0.792414, 1.570796, 1.658814],accel_mss,speed_ms,0,blend_radius_m)
    |   movel([0.088177, -1.291786, -2.627966, -0.792637, 1.570796, 1.658973],accel_mss,speed_ms,0,blend_radius_m)
    |   movel([0.088520, -1.291368, -2.628210, -0.792810, 1.570796, 1.659316],accel_mss,speed_ms,0,blend_radius_m)
    |   movel([0.088850, -1.291076, -2.628381, -0.792932, 1.570796, 1.659647],accel_mss,speed_ms,0,blend_radius_m)
    |   movel([0.089096, -1.290851, -2.628513, -0.793025, 1.570796, 1.659893],accel_mss,speed_ms,0,blend_radius_m)
    |   movel([0.089150, -1.290478, -2.628730, -0.793180, 1.570796, 1.659946],accel_mss,speed_ms,0,blend_radius_m)
    |   movel([0.088850, -1.290441, -2.628752, -0.793196, 1.570796, 1.659646],accel_mss,speed_ms,0,blend_radius_m)
    |   movel([0.088651, -1.290304, -2.628832, -0.793253, 1.570796, 1.659447],accel_mss,speed_ms,0,blend_radius_m)
    |   movel([0.088309, -1.290383, -2.628786, -0.793220, 1.570796, 1.659105],accel_mss,speed_ms,0,blend_radius_m)
    |   movel([0.087687, -1.290468, -2.628736, -0.793185, 1.570796, 1.658483],accel_mss,speed_ms,0,blend_radius_m)
    |   movel([0.087026, -1.290337, -2.628813, -0.793239, 1.570796, 1.657823],accel_mss,speed_ms,0,blend_radius_m)
    |   movel([0.086481, -1.290048, -2.628981, -0.793360, 1.570796, 1.657277],accel_mss,speed_ms,0,blend_radius_m)
    |   movel([0.086205, -1.289649, -2.629214, -0.793526, 1.570796, 1.657001],accel_mss,speed_ms,0,blend_radius_m)
    |   movel([0.086167, -1.289347, -2.629390, -0.793652, 1.570796, 1.656963],accel_mss,speed_ms,0,blend_radius_m)
    |   movel([0.086235, -1.289031, -2.629574, -0.793784, 1.570796, 1.657032],accel_mss,speed_ms,0,blend_radius_m)
    |   movel([0.086426, -1.288658, -2.629791, -0.793940, 1.570796, 1.657222],accel_mss,speed_ms,0,blend_radius_m)
    |   movel([0.086757, -1.288197, -2.630059, -0.794133, 1.570796, 1.657553],accel_mss,speed_ms,0,blend_radius_m)
    |   movel([0.086981, -1.287956, -2.630199, -0.794234, 1.570796, 1.657777],accel_mss,speed_ms,0,blend_radius_m)
    |   movel([0.087305, -1.287686, -2.630355, -0.794348, 1.570796, 1.658101],accel_mss,speed_ms,0,blend_radius_m)
    |   movel([0.087627, -1.287459, -2.630487, -0.794443, 1.570796, 1.658423],accel_mss,speed_ms,0,blend_radius_m)
    |   movel([0.087930, -1.287270, -2.630596, -0.794522, 1.570796, 1.658726],accel_mss,speed_ms,0,blend_radius_m)
    |   movel([0.088216, -1.287266, -2.630599, -0.794524, 1.570796, 1.659013],accel_mss,speed_ms,0,blend_radius_m)
    |   movel([0.088406, -1.287400, -2.630521, -0.794468, 1.570796, 1.659202],accel_mss,speed_ms,0,blend_radius_m)
    |   movel([0.088248, -1.287057, -2.630720, -0.794612, 1.570796, 1.659044],accel_mss,speed_ms,0,blend_radius_m)
    |   movel([0.088513, -1.286866, -2.630831, -0.794692, 1.570796, 1.659309],accel_mss,speed_ms,0,blend_radius_m)
    |   movel([0.088853, -1.286547, -2.631015, -0.794827, 1.570796, 1.659650],accel_mss,speed_ms,0,blend_radius_m)
    |   movel([0.089467, -1.286118, -2.631263, -0.795007, 1.570796, 1.660263],accel_mss,speed_ms,0,blend_radius_m)
    |   movel([0.090092, -1.285722, -2.631492, -0.795175, 1.570796, 1.660888],accel_mss,speed_ms,0,blend_radius_m)
    |   movel([0.090426, -1.285649, -2.631534, -0.795205, 1.570796, 1.661223],accel_mss,speed_ms,0,blend_radius_m)
    |   movel([0.090517, -1.285894, -2.631393, -0.795102, 1.570796, 1.661314],accel_mss,speed_ms,0,blend_radius_m)
    |   speed_ms = 0.003
    |   movel([0.090517, -1.289419, -2.633037, -0.789932, 1.570796, 1.661314],accel_mss,speed_ms,0,blend_radius_m)
    |   speed_ms = 0.007
    |   movel([0.090760, -1.289481, -2.633001, -0.789907, 1.570796, 1.661556],accel_mss,speed_ms,0,blend_radius_m)
    |   movel([0.091359, -1.289492, -2.632995, -0.789902, 1.570796, 1.662155],accel_mss,speed_ms,0,blend_radius_m)
    |   movel([0.091835, -1.289537, -2.632969, -0.789883, 1.570796, 1.662631],accel_mss,speed_ms,0,blend_radius_m)
    |   movel([0.092380, -1.289595, -2.632935, -0.789859, 1.570796, 1.663177],accel_mss,speed_ms,0,blend_radius_m)
    |   movel([0.092996, -1.289644, -2.632907, -0.789838, 1.570796, 1.663793],accel_mss,speed_ms,0,blend_radius_m)
    |   movel([0.093656, -1.289662, -2.632896, -0.789831, 1.570796, 1.664452],accel_mss,speed_ms,0,blend_radius_m)
    |   movel([0.094270, -1.289652, -2.632902, -0.789835, 1.570796, 1.665066],accel_mss,speed_ms,0,blend_radius_m)
    |   movel([0.094742, -1.289607, -2.632928, -0.789854, 1.570796, 1.665538],accel_mss,speed_ms,0,blend_radius_m)
    |   movel([0.097078, -1.289084, -2.633232, -0.790073, 1.570796, 1.667875],accel_mss,speed_ms,0,blend_radius_m)
    |   movel([0.099439, -1.288210, -2.633739, -0.790440, 1.570796, 1.670236],accel_mss,speed_ms,0,blend_radius_m)
    |   movel([0.101784, -1.287001, -2.634438, -0.790950, 1.570796, 1.672581],accel_mss,speed_ms,0,blend_radius_m)
    |   movel([0.104076, -1.285475, -2.635318, -0.791596, 1.570796, 1.674873],accel_mss,speed_ms,0,blend_radius_m)
    |   movel([0.104777, -1.285009, -2.635587, -0.791794, 1.570796, 1.675573],accel_mss,speed_ms,0,blend_radius_m)
    |   movel([0.105551, -1.284591, -2.635827, -0.791971, 1.570796, 1.676347],accel_mss,speed_ms,0,blend_radius_m)
    |   movel([0.106203, -1.284312, -2.635987, -0.792090, 1.570796, 1.676999],accel_mss,speed_ms,0,blend_radius_m)
    |   movel([0.106394, -1.284460, -2.635902, -0.792027, 1.570796, 1.677190],accel_mss,speed_ms,0,blend_radius_m)
    |   movel([0.106666, -1.284467, -2.635898, -0.792024, 1.570796, 1.677462],accel_mss,speed_ms,0,blend_radius_m)
    |   movel([0.106922, -1.284176, -2.636065, -0.792148, 1.570796, 1.677719],accel_mss,speed_ms,0,blend_radius_m)
    |   movel([0.107235, -1.284090, -2.636114, -0.792184, 1.570796, 1.678032],accel_mss,speed_ms,0,blend_radius_m)
    |   movel([0.106944, -1.284195, -2.636054, -0.792140, 1.570796, 1.677741],accel_mss,speed_ms,0,blend_radius_m)
    |   movel([0.107092, -1.284446, -2.635910, -0.792033, 1.570796, 1.677889],accel_mss,speed_ms,0,blend_radius_m)
    |   movel([0.107397, -1.284361, -2.635959, -0.792069, 1.570796, 1.678194],accel_mss,speed_ms,0,blend_radius_m)
    |   movel([0.107675, -1.284389, -2.635943, -0.792057, 1.570796, 1.678471],accel_mss,speed_ms,0,blend_radius_m)
    |   movel([0.107807, -1.284548, -2.635851, -0.791989, 1.570796, 1.678603],accel_mss,speed_ms,0,blend_radius_m)
    |   movel([0.108113, -1.284359, -2.635960, -0.792070, 1.570796, 1.678910],accel_mss,speed_ms,0,blend_radius_m)
    |   movel([0.107859, -1.284295, -2.635997, -0.792097, 1.570796, 1.678655],accel_mss,speed_ms,0,blend_radius_m)
    |   movel([0.107530, -1.284175, -2.636066, -0.792148, 1.570796, 1.678327],accel_mss,speed_ms,0,blend_radius_m)
    |   movel([0.108087, -1.283955, -2.636192, -0.792242, 1.570796, 1.678883],accel_mss,speed_ms,0,blend_radius_m)
    |   movel([0.108555, -1.283993, -2.636170, -0.792226, 1.570796, 1.679351],accel_mss,speed_ms,0,blend_radius_m)
    |   movel([0.109052, -1.284191, -2.636057, -0.792141, 1.570796, 1.679849],accel_mss,speed_ms,0,blend_radius_m)
    |   movel([0.109447, -1.284471, -2.635896, -0.792022, 1.570796, 1.680244],accel_mss,speed_ms,0,blend_radius_m)
    |   movel([0.109568, -1.284760, -2.635730, -0.791899, 1.570796, 1.680365],accel_mss,speed_ms,0,blend_radius_m)
    |   movel([0.109559, -1.285168, -2.635495, -0.791726, 1.570796, 1.680355],accel_mss,speed_ms,0,blend_radius_m)
    |   movel([0.109485, -1.285459, -2.635327, -0.791602, 1.570796, 1.680281],accel_mss,speed_ms,0,blend_radius_m)
    |   movel([0.109326, -1.285744, -2.635163, -0.791481, 1.570796, 1.680122],accel_mss,speed_ms,0,blend_radius_m)
    |   movel([0.109017, -1.286131, -2.634940, -0.791318, 1.570796, 1.679813],accel_mss,speed_ms,0,blend_radius_m)
    |   movel([0.108778, -1.286389, -2.634792, -0.791209, 1.570796, 1.679574],accel_mss,speed_ms,0,blend_radius_m)
    |   movel([0.108466, -1.286690, -2.634618, -0.791081, 1.570796, 1.679263],accel_mss,speed_ms,0,blend_radius_m)
    |   movel([0.108137, -1.286981, -2.634449, -0.790958, 1.570796, 1.678934],accel_mss,speed_ms,0,blend_radius_m)
    |   movel([0.107842, -1.287219, -2.634312, -0.790858, 1.570796, 1.678638],accel_mss,speed_ms,0,blend_radius_m)
    |   movel([0.107121, -1.287746, -2.634007, -0.790636, 1.570796, 1.677917],accel_mss,speed_ms,0,blend_radius_m)
    |   movel([0.106892, -1.287657, -2.634059, -0.790673, 1.570796, 1.677688],accel_mss,speed_ms,0,blend_radius_m)
    |   movel([0.107390, -1.287075, -2.634396, -0.790919, 1.570796, 1.678187],accel_mss,speed_ms,0,blend_radius_m)
    |   movel([0.107724, -1.286699, -2.634612, -0.791077, 1.570796, 1.678521],accel_mss,speed_ms,0,blend_radius_m)
    |   movel([0.107352, -1.286905, -2.634494, -0.790991, 1.570796, 1.678148],accel_mss,speed_ms,0,blend_radius_m)
    |   movel([0.107190, -1.287198, -2.634325, -0.790867, 1.570796, 1.677986],accel_mss,speed_ms,0,blend_radius_m)
    |   movel([0.106820, -1.287315, -2.634257, -0.790817, 1.570796, 1.677616],accel_mss,speed_ms,0,blend_radius_m)
    |   movel([0.106429, -1.287680, -2.634045, -0.790663, 1.570796, 1.677225],accel_mss,speed_ms,0,blend_radius_m)
    |   movel([0.106409, -1.287958, -2.633885, -0.790546, 1.570796, 1.677205],accel_mss,speed_ms,0,blend_radius_m)
    |   movel([0.106162, -1.287866, -2.633938, -0.790585, 1.570796, 1.676958],accel_mss,speed_ms,0,blend_radius_m)
    |   movel([0.105915, -1.288217, -2.633735, -0.790437, 1.570796, 1.676711],accel_mss,speed_ms,0,blend_radius_m)
    |   movel([0.106042, -1.288507, -2.633567, -0.790315, 1.570796, 1.676838],accel_mss,speed_ms,0,blend_radius_m)
    |   movel([0.106016, -1.288793, -2.633401, -0.790195, 1.570796, 1.676812],accel_mss,speed_ms,0,blend_radius_m)
    |   movel([0.106280, -1.288784, -2.633406, -0.790199, 1.570796, 1.677077],accel_mss,speed_ms,0,blend_radius_m)
    |   movel([0.106205, -1.289096, -2.633225, -0.790068, 1.570796, 1.677002],accel_mss,speed_ms,0,blend_radius_m)
    |   movel([0.106244, -1.289354, -2.633075, -0.789960, 1.570796, 1.677041],accel_mss,speed_ms,0,blend_radius_m)
    |   movel([0.106515, -1.289523, -2.632977, -0.789889, 1.570796, 1.677311],accel_mss,speed_ms,0,blend_radius_m)
    |   movel([0.106800, -1.289339, -2.633084, -0.789966, 1.570796, 1.677596],accel_mss,speed_ms,0,blend_radius_m)
    |   movel([0.106483, -1.289380, -2.633060, -0.789949, 1.570796, 1.677280],accel_mss,speed_ms,0,blend_radius_m)
    |   movel([0.106363, -1.289102, -2.633221, -0.790065, 1.570796, 1.677160],accel_mss,speed_ms,0,blend_radius_m)
    |   movel([0.106782, -1.288931, -2.633321, -0.790137, 1.570796, 1.677578],accel_mss,speed_ms,0,blend_radius_m)
    |   movel([0.106980, -1.289067, -2.633242, -0.790080, 1.570796, 1.677777],accel_mss,speed_ms,0,blend_radius_m)
    |   movel([0.107145, -1.289309, -2.633101, -0.789979, 1.570796, 1.677941],accel_mss,speed_ms,0,blend_radius_m)
    |   movel([0.107185, -1.289603, -2.632931, -0.789856, 1.570796, 1.677981],accel_mss,speed_ms,0,blend_radius_m)
    |   movel([0.107094, -1.289907, -2.632754, -0.789728, 1.570796, 1.677891],accel_mss,speed_ms,0,blend_radius_m)
    |   movel([0.106889, -1.290184, -2.632593, -0.789612, 1.570796, 1.677685],accel_mss,speed_ms,0,blend_radius_m)
    |   movel([0.106730, -1.290544, -2.632383, -0.789462, 1.570796, 1.677527],accel_mss,speed_ms,0,blend_radius_m)
    |   movel([0.106361, -1.290960, -2.632141, -0.789288, 1.570796, 1.677157],accel_mss,speed_ms,0,blend_radius_m)
    |   movel([0.106023, -1.291272, -2.631959, -0.789158, 1.570796, 1.676819],accel_mss,speed_ms,0,blend_radius_m)
    |   movel([0.105735, -1.291485, -2.631835, -0.789069, 1.570796, 1.676531],accel_mss,speed_ms,0,blend_radius_m)
    |   movel([0.105337, -1.291671, -2.631726, -0.788992, 1.570796, 1.676133],accel_mss,speed_ms,0,blend_radius_m)
    |   movel([0.104955, -1.291907, -2.631589, -0.788894, 1.570796, 1.675752],accel_mss,speed_ms,0,blend_radius_m)
    |   movel([0.104548, -1.292105, -2.631472, -0.788811, 1.570796, 1.675345],accel_mss,speed_ms,0,blend_radius_m)
    |   movel([0.103748, -1.292296, -2.631361, -0.788732, 1.570796, 1.674544],accel_mss,speed_ms,0,blend_radius_m)
    |   movel([0.103011, -1.292524, -2.631228, -0.788637, 1.570796, 1.673807],accel_mss,speed_ms,0,blend_radius_m)
